C03626=1136.287,55.628,-52.348,-179.813,6.522,149.136
C03627=1136.292,55.380,-52.331,-179.816,6.520,149.137
C03628=1136.297,55.129,-52.315,-179.818,6.519,149.137
C03629=1136.302,54.880,-52.300,-179.821,6.518,149.138
C03630=1136.307,54.631,-52.285,-179.824,6.516,149.138
C03631=1136.312,54.381,-52.269,-179.826,6.515,149.139
C03632=1136.317,54.132,-52.253,-179.829,6.514,149.139
C03633=1136.322,53.883,-52.237,-179.831,6.513,149.140
C03634=1136.327,53.613,-52.220,-179.834,6.512,149.140
C03635=1136.333,53.345,-52.203,-179.837,6.510,149.141
C03636=1136.338,53.076,-52.187,-179.840,6.509,149.142
C03637=1136.343,52.808,-52.170,-179.843,6.507,149.142
C03638=1136.349,52.558,-52.154,-179.846,6.507,149.143
C03639=1136.353,52.309,-52.138,-179.848,6.505,149.143
C03640=1136.358,52.059,-52.122,-179.850,6.504,149.144
C03641=1136.363,51.810,-52.107,-179.854,6.503,149.144
C03642=1136.369,51.561,-52.091,-179.856,6.502,149.145
C03643=1136.373,51.311,-52.075,-179.859,6.500,149.145
C03644=1136.379,51.061,-52.060,-179.862,6.499,149.146
C03645=1136.383,50.812,-52.045,-179.864,6.498,149.146
C03646=1136.388,50.562,-52.029,-179.867,6.497,149.147
C03647=1136.394,50.313,-52.013,-179.869,6.496,149.147
C03648=1136.399,50.063,-51.998,-179.872,6.495,149.148
C03649=1136.404,49.814,-51.983,-179.874,6.494,149.148
C03650=1136.408,49.564,-51.967,-179.878,6.492,149.149
C03651=1136.414,49.315,-51.951,-179.880,6.491,149.149
C03652=1136.418,49.066,-51.936,-179.882,6.490,149.150
C03653=1136.424,48.816,-51.921,-179.885,6.488,149.150
C03654=1136.429,48.567,-51.905,-179.888,6.488,149.151
C03655=1136.433,48.317,-51.890,-179.891,6.486,149.151
C03656=1136.439,48.068,-51.874,-179.893,6.485,149.152
C03657=1136.444,47.818,-51.858,-179.896,6.484,149.152
C03658=1136.449,47.569,-51.843,-179.898,6.483,149.153
C03659=1136.453,47.319,-51.828,-179.901,6.482,149.153
C03660=1136.459,47.070,-51.812,-179.904,6.480,149.154
C03661=1136.463,46.821,-51.797,-179.906,6.480,149.154
C03662=1136.469,46.571,-51.781,-179.909,6.478,149.155
C03663=1136.473,46.322,-51.766,-179.912,6.478,149.156
C03664=1136.479,46.073,-51.751,-179.915,6.476,149.156
C03665=1136.484,45.822,-51.736,-179.917,6.475,149.156
C03666=1136.489,45.573,-51.721,-179.919,6.473,149.157
C03667=1136.494,45.324,-51.705,-179.922,6.473,149.158
C03668=1136.499,45.074,-51.690,-179.925,6.471,149.158
C03669=1136.504,44.825,-51.674,-179.927,6.470,149.158
C03670=1136.509,44.576,-51.659,-179.930,6.469,149.159
C03671=1136.514,44.325,-51.644,-179.932,6.468,149.160
C03672=1136.519,44.076,-51.629,-179.935,6.467,149.160
C03673=1136.524,43.827,-51.614,-179.938,6.466,149.161
C03674=1136.529,43.577,-51.598,-179.941,6.465,149.161
C03675=1136.534,43.328,-51.583,-179.943,6.464,149.162
C03676=1136.540,43.078,-51.568,-179.946,6.463,149.162
C03677=1136.544,42.829,-51.553,-179.949,6.461,149.163
C03678=1136.549,42.579,-51.537,-179.951,6.460,149.163
C03679=1136.554,42.330,-51.522,-179.954,6.459,149.164
C03680=1136.559,42.080,-51.507,-179.956,6.458,149.164
C03681=1136.564,41.831,-51.492,-179.959,6.456,149.165
C03682=1136.569,41.581,-51.477,-179.962,6.456,149.165
C03683=1136.574,41.332,-51.462,-179.964,6.454,149.166
C03684=1136.580,41.082,-51.447,-179.967,6.454,149.166
C03685=1136.584,40.833,-51.432,-179.970,6.452,149.167
C03686=1136.590,40.583,-51.417,-179.972,6.451,149.167
C03687=1136.595,40.334,-51.402,-179.975,6.450,149.168
C03688=1136.600,40.085,-51.386,-179.977,6.449,149.169
C03689=1136.605,39.835,-51.372,-179.980,6.448,149.169
C03690=1136.610,39.585,-51.356,-179.982,6.447,149.169
C03691=1136.614,39.336,-51.341,-179.985,6.445,149.170
C03692=1136.619,39.086,-51.327,-179.988,6.445,149.171
C03693=1136.625,38.837,-51.311,-179.990,6.444,149.171
C03694=1136.630,38.587,-51.297,-179.993,6.442,149.171
C03695=1136.635,38.338,-51.281,-179.995,6.442,149.172
C03696=1136.640,38.088,-51.266,-179.998,6.440,149.173
C03697=1136.645,37.839,-51.252,180.000,6.439,149.173
C03698=1136.650,37.589,-51.237,179.996,6.438,149.174
C03699=1136.655,37.340,-51.222,179.994,6.437,149.174
C03700=1136.660,37.090,-51.207,179.992,6.436,149.175
C03701=1136.665,36.841,-51.192,179.989,6.435,149.175
C03702=1136.670,36.591,-51.177,179.986,6.434,149.176
C03703=1136.676,36.341,-51.163,179.984,6.433,149.176
C03704=1136.680,36.092,-51.148,179.981,6.432,149.177
C03705=1136.685,35.843,-51.133,179.979,6.431,149.177
C03706=1136.691,35.593,-51.118,179.976,6.429,149.178
C03707=1136.696,35.343,-51.103,179.973,6.429,149.178
C03708=1136.700,35.094,-51.088,179.970,6.427,149.179
C03709=1136.706,34.844,-51.074,179.968,6.426,149.179
C03710=1136.711,34.595,-51.059,179.966,6.426,149.180
C03711=1136.716,34.346,-51.044,179.963,6.424,149.180
C03712=1136.721,34.096,-51.029,179.961,6.423,149.181
C03713=1136.726,33.846,-51.014,179.957,6.422,149.182
C03714=1136.731,33.597,-51.000,179.955,6.421,149.182
C03715=1136.736,33.348,-50.985,179.952,6.420,149.183
C03716=1136.742,33.098,-50.971,179.950,6.419,149.183
C03717=1136.747,32.849,-50.956,179.947,6.418,149.184
C03718=1136.751,32.600,-50.941,179.945,6.417,149.184
C03719=1136.756,32.350,-50.927,179.942,6.416,149.185
C03720=1136.762,32.100,-50.912,179.939,6.415,149.185
C03721=1136.767,31.851,-50.897,179.937,6.414,149.186
C03722=1136.772,31.601,-50.883,179.934,6.413,149.186
C03723=1136.777,31.351,-50.869,179.932,6.412,149.187
C03724=1136.782,31.102,-50.853,179.929,6.411,149.187
C03725=1136.787,30.852,-50.839,179.926,6.410,149.188
C03726=1136.792,30.602,-50.825,179.924,6.409,149.188
C03727=1136.797,30.353,-50.810,179.921,6.408,149.189
C03728=1136.802,30.104,-50.796,179.919,6.407,149.190
C03729=1136.808,29.854,-50.781,179.916,6.405,149.190
C03730=1136.813,29.605,-50.767,179.914,6.405,149.191
C03731=1136.817,29.356,-50.752,179.911,6.403,149.191
C03732=1136.822,29.106,-50.737,179.909,6.402,149.192
C03733=1136.827,28.856,-50.723,179.906,6.402,149.192
C03734=1136.832,28.606,-50.709,179.903,6.400,149.193
C03735=1136.837,28.357,-50.694,179.901,6.399,149.193
C03736=1136.843,28.108,-50.679,179.898,6.398,149.194
C03737=1136.848,27.858,-50.665,179.896,6.397,149.194
C03738=1136.853,27.590,-50.649,179.893,6.396,149.195
C03739=1136.859,27.320,-50.634,179.890,6.395,149.195
C03740=1136.864,27.051,-50.619,179.887,6.394,149.196
C03741=1136.870,26.782,-50.602,179.885,6.393,149.197
C03742=1136.875,26.532,-50.588,179.882,6.392,149.197
C03743=1136.880,26.283,-50.574,179.879,6.391,149.198
C03744=1136.885,26.034,-50.560,179.877,6.390,149.198
C03745=1136.890,25.784,-50.545,179.874,6.389,149.199
C03746=1136.895,25.534,-50.531,179.872,6.388,149.199
C03747=1136.900,25.285,-50.517,179.869,6.387,149.200
C03748=1136.905,25.035,-50.503,179.866,6.386,149.200
C03749=1136.911,24.786,-50.489,179.864,6.385,149.201
C03750=1136.916,24.536,-50.474,179.861,6.384,149.201
C03751=1136.921,24.286,-50.460,179.859,6.383,149.202
C03752=1136.925,24.037,-50.445,179.856,6.382,149.202
C03753=1136.930,23.788,-50.431,179.854,6.381,149.203
C03754=1136.936,23.539,-50.417,179.851,6.381,149.204
C03755=1136.941,23.289,-50.403,179.848,6.379,149.204
C03756=1136.946,23.039,-50.388,179.846,6.378,149.205
C03757=1136.951,22.790,-50.374,179.843,6.377,149.205
C03758=1136.956,22.541,-50.360,179.841,6.376,149.206
C03759=1136.961,22.291,-50.346,179.839,6.375,149.206
C03760=1136.966,22.041,-50.332,179.835,6.374,149.207
C03761=1136.971,21.791,-50.317,179.833,6.373,149.207
C03762=1136.977,21.542,-50.304,179.831,6.372,149.208
C03763=1136.982,21.292,-50.290,179.828,6.371,149.208
C03764=1136.987,21.042,-50.276,179.826,6.370,149.209
C03765=1136.992,20.793,-50.261,179.823,6.369,149.209
C03766=1136.997,20.544,-50.247,179.820,6.368,149.210
C03767=1137.002,20.294,-50.233,179.818,6.367,149.210
C03768=1137.007,20.044,-50.219,179.815,6.366,149.211
C03769=1137.013,19.795,-50.205,179.813,6.365,149.212
C03770=1137.018,19.546,-50.191,179.810,6.365,149.212
C03771=1137.023,19.296,-50.176,179.807,6.363,149.213
C03772=1137.027,19.046,-50.163,179.805,6.362,149.213
C03773=1137.033,18.797,-50.150,179.803,6.362,149.214
C03774=1137.038,18.547,-50.135,179.800,6.360,149.214
C03775=1137.043,18.297,-50.121,179.797,6.360,149.215
C03776=1137.048,18.048,-50.107,179.795,6.359,149.215
C03777=1137.053,17.799,-50.093,179.792,6.358,149.216
C03778=1137.058,17.549,-50.079,179.790,6.357,149.216
C03779=1137.064,17.299,-50.065,179.788,6.356,149.217
C03780=1137.068,17.050,-50.052,179.784,6.355,149.218
C03781=1137.073,16.800,-50.037,179.782,6.354,149.218
C03782=1137.079,16.551,-50.024,179.780,6.353,149.219
C03783=1137.084,16.301,-50.009,179.777,6.352,149.219
C03784=1137.089,16.051,-49.996,179.775,6.351,149.220
C03785=1137.094,15.802,-49.982,179.772,6.351,149.220
C03786=1137.099,15.553,-49.968,179.769,6.349,149.221
C03787=1137.104,15.302,-49.955,179.767,6.348,149.221
C03788=1137.109,15.053,-49.941,179.764,6.348,149.222
C03789=1137.114,14.804,-49.926,179.762,6.346,149.222
C03790=1137.119,14.554,-49.912,179.759,6.345,149.223
C03791=1137.125,14.305,-49.899,179.757,6.345,149.223
C03792=1137.129,14.055,-49.885,179.754,6.343,149.224
C03793=1137.135,13.806,-49.871,179.752,6.342,149.224
C03794=1137.140,13.556,-49.858,179.749,6.342,149.225
C03795=1137.145,13.306,-49.844,179.747,6.341,149.226
C03796=1137.150,13.057,-49.830,179.744,6.340,149.226
C03797=1137.155,12.807,-49.817,179.742,6.339,149.227
C03798=1137.161,12.558,-49.803,179.739,6.338,149.227
C03799=1137.165,12.308,-49.789,179.736,6.337,149.228
C03800=1137.170,12.058,-49.775,179.734,6.336,149.228
C03801=1137.176,11.809,-49.761,179.732,6.336,149.229
C03802=1137.180,11.559,-49.749,179.729,6.334,149.229
C03803=1137.186,11.310,-49.735,179.726,6.333,149.230
C03804=1137.191,11.060,-49.720,179.724,6.333,149.230
C03805=1137.197,10.811,-49.707,179.722,6.332,149.231
C03806=1137.201,10.561,-49.693,179.719,6.331,149.232
C03807=1137.206,10.311,-49.680,179.716,6.330,149.232
C03808=1137.212,10.062,-49.666,179.714,6.329,149.233
C03809=1137.216,9.812,-49.653,179.711,6.328,149.233
C03810=1137.222,9.563,-49.639,179.709,6.327,149.234
C03811=1137.227,9.313,-49.626,179.706,6.327,149.234
C03812=1137.232,9.064,-49.612,179.704,6.326,149.235
C03813=1137.237,8.814,-49.599,179.701,6.325,149.235
C03814=1137.243,8.565,-49.585,179.699,6.324,149.236
C03815=1137.247,8.315,-49.572,179.697,6.323,149.236
C03816=1137.253,8.066,-49.558,179.693,6.322,149.237
C03817=1137.257,7.816,-49.545,179.691,6.321,149.237
C03818=1137.263,7.567,-49.531,179.688,6.320,149.238
C03819=1137.268,7.316,-49.517,179.686,6.320,149.239
C03820=1137.273,7.068,-49.504,179.684,6.318,149.239
C03821=1137.278,6.817,-49.491,179.681,6.318,149.240
C03822=1137.283,6.568,-49.478,179.679,6.317,149.240
C03823=1137.288,6.318,-49.464,179.677,6.316,149.241
C03824=1137.294,6.069,-49.450,179.673,6.315,149.241
C03825=1137.298,5.819,-49.437,179.671,6.314,149.242
C03826=1137.304,5.570,-49.424,179.669,6.313,149.242
C03827=1137.309,5.319,-49.411,179.666,6.313,149.243
C03828=1137.314,5.070,-49.397,179.664,6.311,149.243
C03829=1137.319,4.820,-49.384,179.661,6.311,149.244
C03830=1137.325,4.571,-49.371,179.659,6.310,149.245
C03831=1137.329,4.321,-49.357,179.657,6.309,149.245
C03832=1137.335,4.072,-49.344,179.653,6.308,149.246
C03833=1137.339,3.822,-49.331,179.651,6.307,149.246
C03834=1137.345,3.573,-49.317,179.649,6.306,149.247
C03835=1137.350,3.323,-49.304,179.646,6.306,149.247
C03836=1137.355,3.073,-49.291,179.643,6.304,149.248
C03837=1137.360,2.824,-49.277,179.641,6.303,149.248
C03838=1137.365,2.574,-49.264,179.639,6.303,149.249
C03839=1137.371,2.325,-49.251,179.636,6.302,149.249
C03840=1137.376,2.074,-49.238,179.633,6.301,149.250
C03841=1137.381,1.826,-49.224,179.631,6.300,149.251
C03842=1137.386,1.556,-49.210,179.629,6.299,149.251
C03843=1137.393,1.286,-49.196,179.626,6.298,149.252
C03844=1137.397,1.017,-49.182,179.623,6.298,149.252
C03845=1137.403,0.747,-49.167,179.621,6.297,149.253
C03846=1137.408,0.498,-49.155,179.618,6.295,149.253
C03847=1137.413,0.248,-49.141,179.615,6.295,149.254
C03848=1137.418,-0.001,-49.128,179.613,6.294,149.255
C03849=1137.424,-0.251,-49.115,179.610,6.294,149.255
C03850=1137.429,-0.501,-49.102,179.608,6.293,149.256
C03851=1137.434,-0.750,-49.089,179.606,6.291,149.256
C03852=1137.440,-1.000,-49.076,179.603,6.291,149.257
C03853=1137.444,-1.249,-49.062,179.601,6.290,149.257
C03854=1137.450,-1.499,-49.049,179.599,6.289,149.258
C03855=1137.454,-1.749,-49.036,179.595,6.288,149.258
C03856=1137.459,-1.998,-49.024,179.593,6.287,149.259
C03857=1137.465,-2.248,-49.010,179.591,6.286,149.259
C03858=1137.470,-2.498,-48.997,179.588,6.286,149.260
C03859=1137.475,-2.747,-48.985,179.586,6.285,149.261
C03860=1137.481,-2.997,-48.972,179.583,6.284,149.261
C03861=1137.485,-3.247,-48.959,179.581,6.283,149.262
C03862=1137.491,-3.496,-48.945,179.578,6.282,149.262
C03863=1137.496,-3.745,-48.932,179.576,6.282,149.263
C03864=1137.501,-3.995,-48.919,179.574,6.281,149.263
C03865=1137.506,-4.244,-48.907,179.571,6.280,149.264
C03866=1137.512,-4.494,-48.893,179.568,6.279,149.265
C03867=1137.517,-4.743,-48.881,179.566,6.278,149.265
C03868=1137.521,-4.993,-48.868,179.564,6.278,149.265
C03869=1137.527,-5.243,-48.855,179.561,6.277,149.266
C03870=1137.532,-5.492,-48.842,179.559,6.276,149.267
C03871=1137.537,-5.742,-48.829,179.556,6.275,149.267
C03872=1137.543,-5.992,-48.816,179.554,6.274,149.268
C03873=1137.548,-6.241,-48.803,179.551,6.273,149.268
C03874=1137.553,-6.491,-48.791,179.549,6.273,149.269
C03875=1137.557,-6.741,-48.778,179.547,6.272,149.269
C03876=1137.563,-6.990,-48.764,179.544,6.271,149.270
C03877=1137.569,-7.240,-48.753,179.541,6.270,149.271
C03878=1137.573,-7.490,-48.740,179.539,6.269,149.271
C03879=1137.578,-7.739,-48.727,179.537,6.269,149.271
C03880=1137.584,-7.989,-48.714,179.534,6.268,149.272
C03881=1137.589,-8.238,-48.701,179.532,6.267,149.273
C03882=1137.594,-8.488,-48.688,179.529,6.267,149.273
C03883=1137.599,-8.738,-48.676,179.526,6.265,149.274
C03884=1137.604,-8.987,-48.663,179.524,6.265,149.274
C03885=1137.610,-9.237,-48.650,179.522,6.264,149.275
C03886=1137.614,-9.487,-48.637,179.519,6.263,149.275
C03887=1137.620,-9.737,-48.625,179.517,6.263,149.276
C03888=1137.625,-9.986,-48.612,179.515,6.262,149.277
C03889=1137.630,-10.235,-48.600,179.512,6.261,149.277
C03890=1137.635,-10.485,-48.587,179.510,6.260,149.278
C03891=1137.640,-10.735,-48.574,179.507,6.259,149.278
C03892=1137.646,-10.984,-48.561,179.505,6.259,149.279
C03893=1137.651,-11.234,-48.549,179.502,6.258,149.279
C03894=1137.656,-11.483,-48.537,179.500,6.257,149.280
C03895=1137.661,-11.733,-48.524,179.498,6.257,149.280
C03896=1137.666,-11.983,-48.511,179.495,6.255,149.281
C03897=1137.671,-12.232,-48.498,179.492,6.255,149.281
C03898=1137.677,-12.482,-48.486,179.490,6.254,149.282
C03899=1137.682,-12.732,-48.473,179.488,6.253,149.283
C03900=1137.687,-12.981,-48.461,179.485,6.253,149.283
C03901=1137.692,-13.231,-48.448,179.483,6.252,149.284
C03902=1137.697,-13.481,-48.436,179.480,6.251,149.284
C03903=1137.702,-13.730,-48.423,179.478,6.251,149.285
C03904=1137.708,-13.980,-48.411,179.476,6.249,149.285
C03905=1137.713,-14.230,-48.399,179.473,6.249,149.286
C03906=1137.718,-14.479,-48.386,179.471,6.248,149.286
C03907=1137.723,-14.728,-48.374,179.468,6.247,149.287
C03908=1137.728,-14.979,-48.361,179.466,6.247,149.288
C03909=1137.733,-15.228,-48.349,179.464,6.246,149.288
C03910=1137.739,-15.478,-48.335,179.461,6.245,149.289
C03911=1137.744,-15.728,-48.324,179.459,6.245,149.289
C03912=1137.750,-15.977,-48.311,179.456,6.243,149.290
C03913=1137.755,-16.226,-48.298,179.453,6.243,149.290
C03914=1137.760,-16.476,-48.287,179.451,6.242,149.291
C03915=1137.765,-16.726,-48.274,179.449,6.241,149.291
C03916=1137.770,-16.976,-48.261,179.446,6.241,149.292
C03917=1137.775,-17.226,-48.249,179.444,6.240,149.292
C03918=1137.780,-17.475,-48.236,179.442,6.239,149.293
C03919=1137.786,-17.725,-48.225,179.439,6.239,149.294
C03920=1137.791,-17.974,-48.212,179.437,6.238,149.294
C03921=1137.796,-18.223,-48.199,179.434,6.237,149.295
C03922=1137.801,-18.473,-48.188,179.432,6.236,149.295
C03923=1137.807,-18.723,-48.175,179.430,6.235,149.296
C03924=1137.812,-18.973,-48.163,179.427,6.235,149.296
C03925=1137.817,-19.222,-48.150,179.425,6.234,149.297
C03926=1137.823,-19.472,-48.139,179.422,6.233,149.297
C03927=1137.827,-19.722,-48.126,179.420,6.233,149.298
C03928=1137.832,-19.972,-48.114,179.418,6.232,149.299
C03929=1137.837,-20.221,-48.102,179.415,6.231,149.299
C03930=1137.842,-20.471,-48.090,179.413,6.231,149.300
C03931=1137.847,-20.720,-48.077,179.411,6.230,149.300
C03932=1137.853,-20.970,-48.065,179.408,6.229,149.301
C03933=1137.858,-21.219,-48.053,179.405,6.228,149.301
C03934=1137.863,-21.469,-48.041,179.403,6.227,149.302
C03935=1137.869,-21.719,-48.028,179.400,6.227,149.302
C03936=1137.874,-21.969,-48.016,179.398,6.226,149.303
C03937=1137.879,-22.218,-48.004,179.396,6.225,149.303
C03938=1137.885,-22.468,-47.992,179.393,6.225,149.304
C03939=1137.890,-22.718,-47.980,179.391,6.224,149.305
C03940=1137.894,-22.967,-47.968,179.389,6.223,149.305
C03941=1137.900,-23.217,-47.956,179.386,6.223,149.306
C03942=1137.905,-23.466,-47.943,179.384,6.222,149.306
C03943=1137.910,-23.716,-47.932,179.382,6.221,149.307
C03944=1137.916,-23.966,-47.920,179.379,6.221,149.307
C03945=1137.921,-24.215,-47.907,179.377,6.220,149.308
C03946=1137.926,-24.486,-47.894,179.374,6.219,149.309
C03947=1137.932,-24.755,-47.882,179.372,6.218,149.309
C03948=1137.937,-25.026,-47.869,179.369,6.217,149.310
C03949=1137.943,-25.296,-47.855,179.367,6.217,149.310
C03950=1137.948,-25.545,-47.843,179.364,6.216,149.311
C03951=1137.954,-25.794,-47.831,179.362,6.215,149.311
C03952=1137.959,-26.044,-47.820,179.360,6.215,149.312
C03953=1137.965,-26.294,-47.808,179.356,6.213,149.313
C03954=1137.969,-26.543,-47.796,179.354,6.213,149.313
C03955=1137.975,-26.793,-47.784,179.352,6.212,149.314
C03956=1137.980,-27.043,-47.772,179.349,6.212,149.314
C03957=1137.985,-27.293,-47.759,179.347,6.211,149.315
C03958=1137.991,-27.542,-47.747,179.345,6.210,149.315
C03959=1137.995,-27.792,-47.736,179.342,6.210,149.316
C03960=1138.001,-28.042,-47.724,179.340,6.209,149.316
C03961=1138.006,-28.291,-47.712,179.338,6.208,149.317
C03962=1138.011,-28.541,-47.700,179.335,6.208,149.318
C03963=1138.016,-28.791,-47.688,179.333,6.207,149.318
C03964=1138.021,-29.041,-47.677,179.331,6.206,149.318
C03965=1138.026,-29.290,-47.664,179.328,6.206,149.319
C03966=1138.031,-29.540,-47.653,179.326,6.205,149.320
C03967=1138.037,-29.790,-47.641,179.324,6.204,149.320
C03968=1138.043,-30.039,-47.629,179.321,6.204,149.321
C03969=1138.048,-30.289,-47.617,179.319,6.203,149.321
C03970=1138.053,-30.539,-47.606,179.317,6.202,149.322
C03971=1138.058,-30.788,-47.594,179.314,6.202,149.322
C03972=1138.063,-31.038,-47.582,179.312,6.201,149.323
C03973=1138.068,-31.287,-47.570,179.310,6.200,149.323
C03974=1138.073,-31.537,-47.558,179.307,6.200,149.324
C03975=1138.079,-31.787,-47.547,179.305,6.199,149.325
C03976=1138.083,-32.037,-47.535,179.303,6.198,149.325
C03977=1138.090,-32.286,-47.524,179.300,6.198,149.326
C03978=1138.095,-32.535,-47.511,179.298,6.197,149.326
C03979=1138.099,-32.785,-47.500,179.296,6.196,149.327
C03980=1138.105,-33.035,-47.488,179.293,6.196,149.327
C03981=1138.110,-33.285,-47.476,179.291,6.195,149.328
C03982=1138.115,-33.535,-47.465,179.288,6.195,149.329
C03983=1138.120,-33.785,-47.453,179.286,6.194,149.329
C03984=1138.126,-34.034,-47.441,179.284,6.193,149.330
C03985=1138.131,-34.283,-47.430,179.281,6.193,149.330
C03986=1138.136,-34.533,-47.418,179.279,6.192,149.331
C03987=1138.141,-34.783,-47.407,179.277,6.191,149.331
C03988=1138.147,-35.033,-47.395,179.274,6.191,149.332
C03989=1138.152,-35.283,-47.383,179.272,6.190,149.332
C03990=1138.157,-35.532,-47.372,179.270,6.189,149.333
C03991=1138.163,-35.782,-47.360,179.267,6.189,149.334
C03992=1138.167,-36.031,-47.349,179.265,6.188,149.334
C03993=1138.173,-36.281,-47.337,179.263,6.187,149.334
C03994=1138.178,-36.531,-47.326,179.260,6.187,149.335
C03995=1138.184,-36.780,-47.314,179.258,6.186,149.336
C03996=1138.189,-37.030,-47.303,179.256,6.185,149.336
C03997=1138.194,-37.280,-47.291,179.253,6.185,149.337
C03998=1138.199,-37.530,-47.279,179.251,6.184,149.337
C03999=1138.204,-37.779,-47.268,179.249,6.183,149.338
C04000=1138.210,-38.028,-47.257,179.247,6.182,149.338
C04001=1138.215,-38.278,-47.245,179.244,6.182,149.339
C04002=1138.220,-38.528,-47.233,179.242,6.181,149.339
C04003=1138.225,-38.778,-47.222,179.240,6.180,149.340
C04004=1138.231,-39.027,-47.211,179.237,6.180,149.341
C04005=1138.236,-39.277,-47.200,179.235,6.179,149.341
C04006=1138.241,-39.527,-47.188,179.232,6.178,149.342
C04007=1138.246,-39.777,-47.177,179.230,6.178,149.342
C04008=1138.252,-40.026,-47.165,179.228,6.177,149.343
C04009=1138.257,-40.276,-47.154,179.225,6.176,149.343
C04010=1138.262,-40.525,-47.142,179.223,6.176,149.344
C04011=1138.267,-40.775,-47.131,179.221,6.175,149.344
C04012=1138.273,-41.025,-47.120,179.218,6.175,149.345
C04013=1138.278,-41.275,-47.109,179.216,6.174,149.346
C04014=1138.283,-41.525,-47.097,179.214,6.173,149.346
C04015=1138.288,-41.774,-47.086,179.211,6.173,149.347
C04016=1138.294,-42.023,-47.074,179.209,6.173,149.347
C04017=1138.299,-42.273,-47.063,179.207,6.172,149.348
C04018=1138.304,-42.523,-47.052,179.205,6.171,149.348
C04019=1138.310,-42.772,-47.041,179.202,6.171,149.349
C04020=1138.314,-43.022,-47.029,179.200,6.170,149.349
C04021=1138.320,-43.272,-47.017,179.198,6.169,149.350
C04022=1138.325,-43.522,-47.007,179.195,6.169,149.351
C04023=1138.331,-43.772,-46.995,179.193,6.168,149.351
C04024=1138.335,-44.021,-46.984,179.191,6.168,149.351
C04025=1138.340,-44.271,-46.973,179.188,6.167,149.352
C04026=1138.346,-44.521,-46.962,179.186,6.166,149.353
C04027=1138.351,-44.770,-46.951,179.184,6.166,149.353
C04028=1138.356,-45.020,-46.939,179.182,6.165,149.354
C04029=1138.362,-45.269,-46.928,179.179,6.164,149.354
C04030=1138.367,-45.519,-46.917,179.177,6.164,149.355
C04031=1138.372,-45.769,-46.905,179.175,6.163,149.355
C04032=1138.378,-46.018,-46.895,179.172,6.162,149.356
C04033=1138.383,-46.268,-46.884,179.170,6.162,149.356
C04034=1138.388,-46.518,-46.872,179.168,6.162,149.357
C04035=1138.393,-46.767,-46.861,179.165,6.161,149.358
C04036=1138.398,-47.018,-46.851,179.163,6.161,149.358
C04037=1138.404,-47.268,-46.839,179.161,6.160,149.359
C04038=1138.409,-47.516,-46.828,179.158,6.159,149.359
C04039=1138.414,-47.767,-46.817,179.156,6.159,149.360
C04040=1138.419,-48.017,-46.805,179.154,6.158,149.360
C04041=1138.425,-48.266,-46.795,179.151,6.157,149.361
C04042=1138.430,-48.516,-46.784,179.149,6.157,149.361
C04043=1138.436,-48.765,-46.772,179.147,6.156,149.362
C04044=1138.441,-49.015,-46.762,179.145,6.155,149.362
C04045=1138.445,-49.265,-46.750,179.143,6.155,149.363
C04046=1138.451,-49.514,-46.740,179.141,6.155,149.364
C04047=1138.456,-49.764,-46.728,179.138,6.154,149.364
C04048=1138.462,-50.013,-46.717,179.136,6.154,149.365
C04049=1138.467,-50.264,-46.707,179.134,6.153,149.365
C04050=1138.472,-50.535,-46.695,179.131,6.152,149.366
C04051=1138.479,-50.805,-46.683,179.129,6.152,149.366
C04052=1138.484,-51.076,-46.670,179.126,6.151,149.367
C04053=1138.489,-51.347,-46.659,179.124,6.150,149.368
C04054=1138.495,-51.596,-46.648,179.122,6.150,149.368
C04055=1138.500,-51.846,-46.637,179.119,6.149,149.369
C04056=1138.506,-52.095,-46.626,179.117,6.149,149.369
C04057=1138.510,-52.345,-46.615,179.115,6.148,149.370
C04058=1138.515,-52.595,-46.605,179.112,6.147,149.370
C04059=1138.522,-52.845,-46.594,179.110,6.147,149.371
C04060=1138.526,-53.095,-46.582,179.107,6.146,149.371
C04061=1138.532,-53.344,-46.572,179.106,6.146,149.372
C04062=1138.537,-53.594,-46.561,179.103,6.145,149.373
C04063=1138.542,-53.844,-46.551,179.101,6.145,149.373
C04064=1138.548,-54.093,-46.539,179.099,6.144,149.374
C04065=1138.553,-54.343,-46.529,179.096,6.144,149.374
C04066=1138.558,-54.593,-46.517,179.094,6.143,149.375
C04067=1138.564,-54.842,-46.507,179.092,6.142,149.375
C04068=1138.569,-55.092,-46.497,179.090,6.141,149.376
C04069=1138.573,-55.342,-46.485,179.088,6.142,149.376
C04070=1138.579,-55.592,-46.475,179.085,6.141,149.377
C04071=1138.584,-55.842,-46.463,179.083,6.140,149.377
C04072=1138.590,-56.091,-46.453,179.080,6.140,149.378
C04073=1138.595,-56.341,-46.442,179.078,6.139,149.379
C04074=1138.600,-56.590,-46.432,179.076,6.138,149.379
C04075=1138.605,-56.840,-46.421,179.074,6.137,149.379
C04076=1138.611,-57.090,-46.411,179.071,6.137,149.380
C04077=1138.616,-57.340,-46.399,179.070,6.137,149.381
C04078=1138.621,-57.589,-46.389,179.067,6.136,149.381
C04079=1138.626,-57.839,-46.379,179.065,6.136,149.382
C04080=1138.631,-58.088,-46.368,179.063,6.135,149.382
C04081=1138.637,-58.339,-46.357,179.060,6.134,149.383
C04082=1138.643,-58.588,-46.346,179.058,6.134,149.383
C04083=1138.647,-58.838,-46.335,179.056,6.133,149.384
C04084=1138.653,-59.088,-46.325,179.054,6.133,149.384
C04085=1138.658,-59.338,-46.314,179.052,6.132,149.385
C04086=1138.663,-59.587,-46.303,179.050,6.132,149.385
C04087=1138.668,-59.837,-46.293,179.047,6.131,149.386
C04088=1138.674,-60.087,-46.283,179.045,6.130,149.387
C04089=1138.680,-60.336,-46.272,179.043,6.130,149.387
C04090=1138.684,-60.586,-46.261,179.040,6.129,149.388
C04091=1138.690,-60.835,-46.251,179.038,6.129,149.388
C04092=1138.695,-61.086,-46.240,179.036,6.129,149.389
C04093=1138.700,-61.335,-46.230,179.034,6.128,149.389
C04094=1138.705,-61.585,-46.219,179.031,6.127,149.390
C04095=1138.711,-61.834,-46.209,179.029,6.127,149.390
C04096=1138.716,-62.085,-46.198,179.027,6.126,149.391
C04097=1138.721,-62.334,-46.188,179.025,6.126,149.392
C04098=1138.727,-62.584,-46.178,179.023,6.126,149.392
C04099=1138.732,-62.833,-46.166,179.020,6.125,149.393
C04100=1138.737,-63.083,-46.156,179.018,6.124,149.393
C04101=1138.742,-63.333,-46.146,179.016,6.124,149.394
C04102=1138.748,-63.583,-46.135,179.013,6.123,149.394
C04103=1138.753,-63.833,-46.125,179.012,6.123,149.395
C04104=1138.758,-64.082,-46.115,179.010,6.122,149.395
C04105=1138.764,-64.332,-46.104,179.007,6.122,149.396
C04106=1138.769,-64.582,-46.093,179.005,6.121,149.396
C04107=1138.774,-64.831,-46.083,179.003,6.120,149.397
C04108=1138.779,-65.081,-46.072,179.001,6.120,149.397
C04109=1138.785,-65.331,-46.062,178.998,6.120,149.398
C04110=1138.790,-65.580,-46.052,178.996,6.119,149.399
C04111=1138.795,-65.831,-46.041,178.994,6.118,149.399
C04112=1138.801,-66.080,-46.031,178.992,6.117,149.399
C04113=1138.806,-66.329,-46.021,178.989,6.117,149.400
C04114=1138.811,-66.580,-46.011,178.987,6.117,149.401
C04115=1138.817,-66.829,-46.001,178.985,6.116,149.401
C04116=1138.822,-67.079,-45.990,178.983,6.116,149.402
C04117=1138.827,-67.328,-45.979,178.980,6.115,149.402
C04118=1138.832,-67.578,-45.969,178.978,6.114,149.403
C04119=1138.837,-67.828,-45.958,178.977,6.114,149.403
C04120=1138.843,-68.078,-45.948,178.974,6.114,149.404
C04121=1138.849,-68.327,-45.938,178.972,6.113,149.405
C04122=1138.853,-68.577,-45.928,178.970,6.113,149.405
C04123=1138.858,-68.827,-45.918,178.967,6.112,149.405
C04124=1138.864,-69.076,-45.908,178.966,6.112,149.406
C04125=1138.869,-69.327,-45.897,178.963,6.111,149.407
C04126=1138.875,-69.576,-45.887,178.961,6.111,149.407
C04127=1138.880,-69.826,-45.877,178.959,6.110,149.408
C04128=1138.886,-70.075,-45.866,178.956,6.109,149.408
C04129=1138.890,-70.325,-45.856,178.954,6.110,149.409
C04130=1138.896,-70.575,-45.847,178.952,6.109,149.409
C04131=1138.902,-70.825,-45.837,178.950,6.108,149.410
C04132=1138.907,-71.075,-45.826,178.948,6.107,149.410
C04133=1138.912,-71.325,-45.816,178.945,6.107,149.411
C04134=1138.918,-71.574,-45.806,178.944,6.107,149.411
C04135=1138.922,-71.824,-45.796,178.941,6.106,149.412
C04136=1138.928,-72.074,-45.786,178.939,6.105,149.412
C04137=1138.933,-72.323,-45.775,178.937,6.105,149.413
C04138=1138.939,-72.573,-45.765,178.935,6.105,149.414
C04139=1138.944,-72.823,-45.755,178.933,6.104,149.414
C04140=1138.949,-73.072,-45.745,178.931,6.104,149.415
C04141=1138.954,-73.322,-45.735,178.928,6.103,149.415
C04142=1138.960,-73.572,-45.725,178.926,6.102,149.416
C04143=1138.965,-73.822,-45.715,178.924,6.102,149.416
C04144=1138.971,-74.072,-45.704,178.922,6.102,149.417
C04145=1138.976,-74.321,-45.695,178.919,6.101,149.417
C04146=1138.981,-74.570,-45.685,178.917,6.101,149.418
C04147=1138.986,-74.821,-45.674,178.915,6.101,149.418
C04148=1138.992,-75.071,-45.665,178.913,6.100,149.419
C04149=1138.997,-75.320,-45.655,178.911,6.099,149.419
C04150=1139.003,-75.570,-45.645,178.908,6.099,149.420
C04151=1139.008,-75.820,-45.634,178.907,6.099,149.421
C04152=1139.013,-76.069,-45.624,178.905,6.098,149.421
C04153=1139.018,-76.319,-45.615,178.902,6.097,149.422
C04154=1139.024,-76.591,-45.603,178.900,6.097,149.422
C04155=1139.030,-76.862,-45.593,178.898,6.096,149.423
C04156=1139.036,-77.134,-45.582,178.895,6.096,149.423
C04157=1139.042,-77.405,-45.571,178.893,6.095,149.424
C04158=1139.047,-77.655,-45.561,178.891,6.095,149.424
C04159=1139.052,-77.904,-45.552,178.889,6.094,149.425
C04160=1139.057,-78.155,-45.541,178.886,6.094,149.426
C04161=1139.063,-78.404,-45.531,178.884,6.093,149.426
C04162=1139.068,-78.653,-45.522,178.882,6.093,149.427
C04163=1139.074,-78.904,-45.512,178.880,6.092,149.427
C04164=1139.079,-79.153,-45.502,178.878,6.092,149.428
C04165=1139.084,-79.402,-45.492,178.875,6.091,149.428
C04166=1139.089,-79.653,-45.482,178.874,6.091,149.429
C04167=1139.095,-79.903,-45.472,178.872,6.090,149.429
C04168=1139.100,-80.152,-45.463,178.869,6.090,149.430
C04169=1139.106,-80.402,-45.453,178.867,6.090,149.430
C04170=1139.111,-80.652,-45.443,178.865,6.089,149.431
C04171=1139.116,-80.901,-45.433,178.863,6.089,149.431
C04172=1139.122,-81.152,-45.423,178.861,6.088,149.432
C04173=1139.126,-81.401,-45.414,178.859,6.088,149.432
C04174=1139.132,-81.651,-45.404,178.856,6.087,149.433
C04175=1139.138,-81.901,-45.394,178.854,6.087,149.434
C04176=1139.143,-82.150,-45.385,178.852,6.086,149.434
C04177=1139.148,-82.399,-45.374,178.850,6.086,149.434
C04178=1139.153,-82.650,-45.365,178.848,6.085,149.435
C04179=1139.159,-82.900,-45.355,178.846,6.085,149.436
C04180=1139.164,-83.150,-45.345,178.843,6.084,149.436
C04181=1139.169,-83.399,-45.336,178.842,6.084,149.437
C04182=1139.175,-83.649,-45.326,178.840,6.083,149.437
C04183=1139.180,-83.898,-45.317,178.837,6.083,149.438
C04184=1139.186,-84.148,-45.306,178.835,6.083,149.438
C04185=1139.191,-84.398,-45.298,178.833,6.082,149.439
C04186=1139.196,-84.648,-45.287,178.831,6.082,149.439
C04187=1139.201,-84.897,-45.277,178.829,6.081,149.440
C04188=1139.207,-85.147,-45.268,178.827,6.081,149.440
C04189=1139.212,-85.397,-45.258,178.824,6.080,149.441
C04190=1139.217,-85.647,-45.249,178.822,6.080,149.441
C04191=1139.223,-85.896,-45.239,178.821,6.080,149.442
C04192=1139.228,-86.146,-45.230,178.819,6.079,149.442
C04193=1139.234,-86.396,-45.219,178.816,6.078,149.443
C04194=1139.239,-86.646,-45.211,178.815,6.078,149.443
C04195=1139.244,-86.896,-45.200,178.812,6.078,149.444
C04196=1139.249,-87.146,-45.191,178.810,6.077,149.445
C04197=1139.255,-87.395,-45.181,178.808,6.076,149.445
C04198=1139.260,-87.645,-45.172,178.806,6.076,149.446
C04199=1139.265,-87.894,-45.162,178.804,6.076,149.446
C04200=1139.271,-88.144,-45.153,178.801,6.075,149.447
C04201=1139.275,-88.394,-45.143,178.800,6.075,149.447
C04202=1139.281,-88.644,-45.134,178.797,6.075,149.448
C04203=1139.287,-88.894,-45.125,178.795,6.074,149.448
C04204=1139.292,-89.143,-45.115,178.794,6.074,149.449
C04205=1139.297,-89.393,-45.106,178.791,6.073,149.449
C04206=1139.303,-89.643,-45.096,178.789,6.073,149.450
C04207=1139.308,-89.892,-45.087,178.787,6.072,149.450
C04208=1139.314,-90.142,-45.076,178.785,6.072,149.451
C04209=1139.319,-90.392,-45.068,178.783,6.071,149.451
C04210=1139.324,-90.642,-45.059,178.781,6.070,149.452
C04211=1139.329,-90.892,-45.048,178.779,6.070,149.452
C04212=1139.334,-91.142,-45.039,178.776,6.070,149.453
C04213=1139.340,-91.391,-45.029,178.774,6.069,149.453
C04214=1139.345,-91.641,-45.020,178.773,6.069,149.454
C04215=1139.350,-91.891,-45.011,178.770,6.069,149.454
C04216=1139.356,-92.141,-45.001,178.768,6.068,149.455
C04217=1139.361,-92.390,-44.992,178.767,6.068,149.455
C04218=1139.367,-92.641,-44.983,178.764,6.068,149.456
C04219=1139.372,-92.890,-44.973,178.762,6.067,149.457
C04220=1139.377,-93.140,-44.964,178.760,6.067,149.457
C04221=1139.383,-93.390,-44.955,178.758,6.066,149.458
C04222=1139.388,-93.639,-44.945,178.756,6.065,149.458
C04223=1139.393,-93.889,-44.935,178.754,6.065,149.459
C04224=1139.399,-94.139,-44.927,178.752,6.065,149.459
C04225=1139.403,-94.388,-44.917,178.749,6.064,149.460
C04226=1139.409,-94.639,-44.907,178.748,6.064,149.460
C04227=1139.415,-94.888,-44.899,178.745,6.064,149.461
C04228=1139.420,-95.138,-44.890,178.743,6.063,149.461
C04229=1139.425,-95.388,-44.879,178.742,6.063,149.462
C04230=1139.431,-95.637,-44.871,178.739,6.062,149.462
C04231=1139.436,-95.887,-44.862,178.737,6.061,149.463
C04232=1139.442,-96.137,-44.853,178.735,6.062,149.463
C04233=1139.447,-96.386,-44.843,178.733,6.061,149.464
C04234=1139.452,-96.636,-44.834,178.731,6.060,149.464
C04235=1139.458,-96.886,-44.825,178.729,6.060,149.465
C04236=1139.463,-97.136,-44.816,178.727,6.059,149.465
C04237=1139.468,-97.385,-44.806,178.725,6.059,149.466
C04238=1139.473,-97.635,-44.797,178.723,6.059,149.466
C04239=1139.479,-97.885,-44.788,178.721,6.058,149.467
C04240=1139.484,-98.135,-44.779,178.719,6.058,149.467
C04241=1139.489,-98.385,-44.770,178.717,6.058,149.468
C04242=1139.495,-98.635,-44.760,178.715,6.057,149.468
C04243=1139.500,-98.884,-44.751,178.713,6.057,149.469
C04244=1139.505,-99.134,-44.742,178.711,6.056,149.469
C04245=1139.511,-99.384,-44.733,178.709,6.055,149.470
C04246=1139.517,-99.634,-44.724,178.707,6.056,149.470
C04247=1139.522,-99.883,-44.715,178.704,6.055,149.471
C04248=1139.527,-100.133,-44.706,178.702,6.054,149.472
C04249=1139.532,-100.382,-44.696,178.700,6.054,149.472
C04250=1139.538,-100.633,-44.687,178.698,6.054,149.473
C04251=1139.543,-100.882,-44.678,178.697,6.054,149.473
C04252=1139.549,-101.132,-44.669,178.694,6.053,149.474
C04253=1139.554,-101.382,-44.660,178.692,6.052,149.474
C04254=1139.560,-101.632,-44.651,178.691,6.052,149.474
C04255=1139.565,-101.882,-44.642,178.688,6.052,149.475
C04256=1139.571,-102.131,-44.633,178.686,6.051,149.476
C04257=1139.576,-102.381,-44.624,178.684,6.051,149.476
C04258=1139.581,-102.653,-44.614,178.682,6.050,149.477
C04259=1139.587,-102.926,-44.605,178.680,6.050,149.477
C04260=1139.592,-103.198,-44.594,178.677,6.049,149.478
C04261=1139.599,-103.470,-44.584,178.676,6.049,149.478
C04262=1139.604,-103.720,-44.575,178.673,6.049,149.479
C04263=1139.610,-103.969,-44.567,178.671,6.048,149.479
C04264=1139.615,-104.219,-44.558,178.670,6.048,149.480
C04265=1139.620,-104.469,-44.549,178.667,6.047,149.480
C04266=1139.625,-104.719,-44.540,178.666,6.047,149.481
C04267=1139.631,-104.969,-44.531,178.663,6.047,149.482
C04268=1139.637,-105.219,-44.522,178.661,6.046,149.482
C04269=1139.642,-105.469,-44.513,178.659,6.046,149.482
C04270=1139.647,-105.718,-44.504,178.657,6.045,149.483
C04271=1139.653,-105.968,-44.495,178.656,6.045,149.483
C04272=1139.658,-106.218,-44.487,178.653,6.045,149.484
C04273=1139.663,-106.468,-44.478,178.651,6.044,149.484
C04274=1139.668,-106.717,-44.469,178.650,6.044,149.485
C04275=1139.673,-106.967,-44.460,178.647,6.043,149.485
C04276=1139.680,-107.217,-44.451,178.646,6.043,149.486
C04277=1139.685,-107.467,-44.442,178.643,6.043,149.487
C04278=1139.690,-107.716,-44.433,178.641,6.042,149.487
C04279=1139.695,-107.966,-44.424,178.639,6.042,149.488
C04280=1139.700,-108.216,-44.415,178.637,6.041,149.488
C04281=1139.706,-108.465,-44.407,178.635,6.041,149.489
C04282=1139.711,-108.715,-44.398,178.633,6.041,149.489
C04283=1139.717,-108.965,-44.389,178.631,6.040,149.490
C04284=1139.722,-109.215,-44.380,178.629,6.040,149.490
C04285=1139.727,-109.465,-44.371,178.627,6.039,149.490
C04286=1139.733,-109.714,-44.363,178.626,6.039,149.491
C04287=1139.738,-109.964,-44.354,178.623,6.039,149.491
C04288=1139.744,-110.214,-44.345,178.621,6.038,149.492
C04289=1139.749,-110.464,-44.336,178.620,6.038,149.492
C04290=1139.754,-110.714,-44.327,178.617,6.038,149.493
C04291=1139.760,-110.963,-44.318,178.615,6.038,149.494
C04292=1139.765,-111.213,-44.310,178.613,6.037,149.494
C04293=1139.770,-111.463,-44.301,178.612,6.037,149.495
C04294=1139.776,-111.714,-44.293,178.609,6.036,149.495
C04295=1139.782,-111.963,-44.284,178.607,6.035,149.496
C04296=1139.787,-112.213,-44.275,178.606,6.035,149.496
C04297=1139.792,-112.462,-44.266,178.603,6.035,149.497
C04298=1139.797,-112.712,-44.257,178.602,6.035,149.497
C04299=1139.803,-112.961,-44.249,178.600,6.034,149.498
C04300=1139.808,-113.212,-44.241,178.597,6.033,149.498
C04301=1139.814,-113.462,-44.232,178.596,6.033,149.499
C04302=1139.819,-113.712,-44.223,178.594,6.032,149.499
C04303=1139.825,-113.961,-44.214,178.592,6.033,149.499
C04304=1139.830,-114.211,-44.206,178.590,6.032,149.500
C04305=1139.835,-114.461,-44.197,178.588,6.032,149.500
C04306=1139.840,-114.711,-44.188,178.586,6.031,149.501
C04307=1139.846,-114.960,-44.180,178.584,6.032,149.502
C04308=1139.851,-115.210,-44.171,178.582,6.031,149.502
C04309=1139.857,-115.460,-44.163,178.580,6.030,149.503
C04310=1139.863,-115.709,-44.154,178.578,6.030,149.503
C04311=1139.868,-115.959,-44.145,178.576,6.029,149.504
C04312=1139.873,-116.210,-44.137,178.574,6.029,149.504
C04313=1139.879,-116.459,-44.129,178.572,6.029,149.505
C04314=1139.883,-116.708,-44.120,178.570,6.029,149.505
C04315=1139.889,-116.958,-44.111,178.568,6.028,149.506
C04316=1139.894,-117.209,-44.103,178.566,6.027,149.506
C04317=1139.900,-117.458,-44.095,178.564,6.027,149.507
C04318=1139.905,-117.708,-44.086,178.562,6.026,149.507
C04319=1139.910,-117.958,-44.078,178.561,6.027,149.508
C04320=1139.916,-118.207,-44.069,178.558,6.026,149.508
C04321=1139.921,-118.457,-44.060,178.557,6.026,149.508
C04322=1139.927,-118.708,-44.052,178.555,6.025,149.509
C04323=1139.933,-118.957,-44.043,178.553,6.025,149.509
C04324=1139.938,-119.207,-44.034,178.551,6.024,149.510
C04325=1139.942,-119.457,-44.027,178.549,6.024,149.510
C04326=1139.948,-119.706,-44.018,178.547,6.024,149.511
C04327=1139.953,-119.956,-44.009,178.545,6.023,149.511
C04328=1139.959,-120.206,-44.001,178.543,6.023,149.512
C04329=1139.965,-120.456,-43.993,178.541,6.022,149.512
C04330=1139.970,-120.705,-43.984,178.539,6.022,149.513
C04331=1139.975,-120.956,-43.976,178.537,6.022,149.513
C04332=1139.981,-121.205,-43.967,178.536,6.022,149.514
C04333=1139.986,-121.455,-43.960,178.533,6.021,149.514
C04334=1139.991,-121.705,-43.951,178.532,6.021,149.515
C04335=1139.997,-121.954,-43.942,178.530,6.020,149.515
C04336=1140.002,-122.205,-43.934,178.528,6.020,149.516
C04337=1140.008,-122.454,-43.925,178.526,6.019,149.516
C04338=1140.013,-122.704,-43.917,178.524,6.019,149.517
C04339=1140.018,-122.954,-43.909,178.522,6.019,149.517
C04340=1140.024,-123.204,-43.901,178.521,6.019,149.518
C04341=1140.029,-123.453,-43.892,178.518,6.018,149.518
C04342=1140.035,-123.704,-43.884,178.516,6.017,149.519
C04343=1140.040,-123.953,-43.875,178.515,6.017,149.519
C04344=1140.045,-124.203,-43.867,178.512,6.017,149.520
C04345=1140.051,-124.452,-43.859,178.511,6.017,149.520
C04346=1140.056,-124.702,-43.850,178.509,6.016,149.521
C04347=1140.061,-124.953,-43.842,178.507,6.016,149.521
C04348=1140.067,-125.202,-43.834,178.505,6.015,149.522
C04349=1140.072,-125.452,-43.826,178.503,6.015,149.522
C04350=1140.078,-125.701,-43.818,178.501,6.014,149.523
C04351=1140.083,-125.952,-43.809,178.499,6.015,149.523
C04352=1140.089,-126.201,-43.801,178.497,6.014,149.524
C04353=1140.094,-126.451,-43.793,178.496,6.014,149.524
C04354=1140.099,-126.701,-43.784,178.493,6.013,149.525
C04355=1140.105,-126.951,-43.777,178.492,6.013,149.525
C04356=1140.110,-127.201,-43.768,178.490,6.012,149.526
C04357=1140.115,-127.450,-43.760,178.488,6.012,149.526
C04358=1140.121,-127.700,-43.752,178.486,6.012,149.527
C04359=1140.127,-127.949,-43.744,178.484,6.012,149.527
C04360=1140.132,-128.200,-43.736,178.482,6.011,149.528
C04361=1140.137,-128.449,-43.727,178.480,6.011,149.528
C04362=1139.716,-128.461,-43.771,178.477,6.014,149.530
C04363=1139.711,-128.210,-43.779,178.479,6.015,149.529
C04364=1139.705,-127.961,-43.788,178.480,6.015,149.529
C04365=1139.700,-127.711,-43.795,178.483,6.016,149.528
C04366=1139.695,-127.462,-43.804,178.484,6.016,149.528
C04367=1139.689,-127.211,-43.812,178.486,6.016,149.527
C04368=1139.684,-126.962,-43.821,178.488,6.016,149.527
C04369=1139.679,-126.712,-43.828,178.490,6.017,149.526
C04370=1139.673,-126.462,-43.837,178.492,6.017,149.526
C04371=1139.667,-126.213,-43.845,178.494,6.018,149.525
C04372=1139.662,-125.963,-43.854,178.495,6.018,149.525
C04373=1139.657,-125.713,-43.861,178.498,6.019,149.524
C04374=1139.652,-125.463,-43.870,178.499,6.019,149.524
C04375=1139.646,-125.213,-43.878,178.501,6.019,149.523
C04376=1139.640,-124.964,-43.886,178.503,6.019,149.523
C04377=1139.635,-124.713,-43.895,178.505,6.020,149.522
C04378=1139.630,-124.464,-43.903,178.507,6.020,149.522
C04379=1139.624,-124.214,-43.911,178.509,6.021,149.522
C04380=1139.619,-123.964,-43.920,178.511,6.021,149.521
C04381=1139.613,-123.714,-43.927,178.513,6.021,149.521
C04382=1139.608,-123.465,-43.936,178.515,6.022,149.520
C04383=1139.603,-123.215,-43.944,178.517,6.022,149.520
C04384=1139.598,-122.965,-43.952,178.519,6.023,149.519
C04385=1139.592,-122.715,-43.961,178.520,6.023,149.519
C04386=1139.586,-122.466,-43.969,178.523,6.023,149.518
C04387=1139.581,-122.215,-43.977,178.524,6.023,149.518
C04388=1139.576,-121.966,-43.986,178.526,6.024,149.517
C04389=1139.571,-121.716,-43.994,178.528,6.024,149.517
C04390=1139.565,-121.466,-44.002,178.530,6.025,149.516
C04391=1139.560,-121.216,-44.011,178.532,6.025,149.516
C04392=1139.554,-120.966,-44.019,178.534,6.026,149.515
C04393=1139.549,-120.716,-44.028,178.536,6.026,149.515
C04394=1139.543,-120.467,-44.037,178.538,6.026,149.514
C04395=1139.538,-120.217,-44.044,178.539,6.026,149.514
C04396=1139.533,-119.967,-44.053,178.542,6.027,149.513
C04397=1139.527,-119.718,-44.062,178.544,6.028,149.513
C04398=1139.522,-119.468,-44.070,178.545,6.028,149.512
C04399=1139.517,-119.218,-44.079,178.548,6.028,149.512
C04400=1139.511,-118.968,-44.086,178.549,6.028,149.511
C04401=1139.505,-118.718,-44.095,178.551,6.029,149.511
C04402=1139.500,-118.468,-44.104,178.553,6.029,149.510
C04403=1139.495,-118.219,-44.111,178.555,6.030,149.510
C04404=1139.490,-117.969,-44.120,178.557,6.030,149.509
C04405=1139.485,-117.719,-44.129,178.559,6.031,149.509
C04406=1139.479,-117.469,-44.137,178.561,6.030,149.508
C04407=1139.473,-117.220,-44.146,178.563,6.031,149.508
C04408=1139.468,-116.970,-44.155,178.565,6.032,149.507
C04409=1139.463,-116.720,-44.164,178.567,6.032,149.507
C04410=1139.457,-116.470,-44.172,178.569,6.033,149.506
C04411=1139.452,-116.220,-44.180,178.570,6.033,149.506
C04412=1139.447,-115.970,-44.189,178.573,6.033,149.505
C04413=1139.441,-115.721,-44.197,178.574,6.033,149.505
C04414=1139.435,-115.471,-44.206,178.576,6.034,149.504
C04415=1139.430,-115.221,-44.215,178.578,6.034,149.504
C04416=1139.424,-114.972,-44.223,178.581,6.034,149.503
C04417=1139.419,-114.721,-44.232,178.583,6.035,149.503
C04418=1139.414,-114.471,-44.241,178.584,6.035,149.502
C04419=1139.409,-114.222,-44.249,178.587,6.036,149.502
C04420=1139.403,-113.973,-44.258,178.588,6.036,149.501
C04421=1139.398,-113.723,-44.267,178.590,6.037,149.501
C04422=1139.392,-113.472,-44.275,178.592,6.037,149.500
C04423=1139.387,-113.222,-44.284,178.594,6.037,149.500
C04424=1139.381,-112.973,-44.293,178.596,6.038,149.499
C04425=1139.376,-112.723,-44.301,178.598,6.038,149.499
C04426=1139.371,-112.473,-44.310,178.600,6.039,149.498
C04427=1139.365,-112.223,-44.318,178.602,6.039,149.498
C04428=1139.360,-111.974,-44.327,178.604,6.039,149.497
C04429=1139.355,-111.724,-44.336,178.606,6.039,149.497
C04430=1139.349,-111.474,-44.345,178.608,6.040,149.496
C04431=1139.344,-111.224,-44.354,178.610,6.041,149.496
C04432=1139.338,-110.975,-44.362,178.612,6.041,149.495
C04433=1139.333,-110.725,-44.370,178.614,6.042,149.495
C04434=1139.328,-110.475,-44.379,178.616,6.041,149.494
C04435=1139.323,-110.225,-44.388,178.618,6.042,149.494
C04436=1139.317,-109.976,-44.397,178.620,6.043,149.493
C04437=1139.312,-109.726,-44.406,178.622,6.043,149.493
C04438=1139.307,-109.476,-44.415,178.624,6.043,149.492
C04439=1139.301,-109.226,-44.423,178.626,6.043,149.492
C04440=1139.296,-108.976,-44.432,178.628,6.044,149.491
C04441=1139.290,-108.727,-44.441,178.630,6.045,149.491
C04442=1139.285,-108.477,-44.449,178.632,6.045,149.490
C04443=1139.280,-108.227,-44.458,178.634,6.046,149.490
C04444=1139.275,-107.977,-44.467,178.635,6.045,149.489
C04445=1139.269,-107.727,-44.476,178.638,6.046,149.489
C04446=1139.263,-107.478,-44.485,178.639,6.046,149.488
C04447=1139.258,-107.228,-44.494,178.642,6.047,149.488
C04448=1139.253,-106.978,-44.503,178.644,6.047,149.487
C04449=1139.247,-106.728,-44.512,178.646,6.047,149.487
C04450=1139.242,-106.478,-44.520,178.648,6.048,149.486
C04451=1139.237,-106.229,-44.529,178.650,6.049,149.486
C04452=1139.231,-105.979,-44.538,178.652,6.049,149.485
C04453=1139.226,-105.730,-44.547,178.654,6.049,149.485
C04454=1139.220,-105.479,-44.556,178.655,6.049,149.484
C04455=1139.215,-105.230,-44.565,178.658,6.050,149.484
C04456=1139.210,-104.980,-44.574,178.660,6.051,149.483
C04457=1139.205,-104.730,-44.583,178.661,6.051,149.483
C04458=1139.199,-104.481,-44.592,178.664,6.051,149.482
C04459=1139.194,-104.231,-44.600,178.666,6.051,149.482
C04460=1139.189,-103.981,-44.609,178.668,6.052,149.481
C04461=1139.183,-103.731,-44.619,178.670,6.053,149.481
C04462=1139.178,-103.481,-44.628,178.672,6.053,149.480
C04463=1139.172,-103.209,-44.638,178.674,6.053,149.480
C04464=1139.166,-102.936,-44.647,178.677,6.054,149.479
C04465=1139.160,-102.665,-44.657,178.679,6.054,149.478
C04466=1139.154,-102.393,-44.667,178.680,6.054,149.478
C04467=1139.149,-102.143,-44.676,178.683,6.055,149.478
C04468=1139.144,-101.893,-44.685,178.685,6.056,149.477
C04469=1139.138,-101.643,-44.694,178.686,6.056,149.477
C04470=1139.133,-101.393,-44.703,178.689,6.056,149.476
C04471=1139.128,-101.143,-44.712,178.691,6.056,149.475
C04472=1139.123,-100.893,-44.721,178.693,6.057,149.475
C04473=1139.117,-100.644,-44.731,178.695,6.058,149.474
C04474=1139.111,-100.395,-44.740,178.697,6.058,149.474
C04475=1139.106,-100.145,-44.748,178.699,6.058,149.473
C04476=1139.101,-99.895,-44.757,178.701,6.059,149.473
C04477=1139.095,-99.645,-44.767,178.703,6.059,149.472
C04478=1139.090,-99.395,-44.776,178.705,6.060,149.472
C04479=1139.085,-99.145,-44.785,178.708,6.060,149.471
C04480=1139.080,-98.896,-44.794,178.709,6.060,149.471
C04481=1139.074,-98.646,-44.804,178.711,6.061,149.470
C04482=1139.069,-98.396,-44.813,178.713,6.061,149.470
C04483=1139.064,-98.146,-44.822,178.715,6.062,149.469
C04484=1139.059,-97.896,-44.830,178.717,6.062,149.469
C04485=1139.052,-97.647,-44.840,178.719,6.062,149.468
C04486=1139.047,-97.397,-44.849,178.721,6.063,149.468
C04487=1139.042,-97.148,-44.858,178.724,6.064,149.467
C04488=1139.036,-96.897,-44.868,178.725,6.064,149.467
C04489=1139.031,-96.648,-44.876,178.728,6.064,149.466
C04490=1139.026,-96.398,-44.886,178.730,6.065,149.466
C04491=1139.020,-96.148,-44.896,178.731,6.065,149.465
C04492=1139.015,-95.898,-44.904,178.734,6.066,149.465
C04493=1139.010,-95.648,-44.913,178.736,6.066,149.464
C04494=1139.004,-95.399,-44.924,178.738,6.066,149.464
C04495=1138.999,-95.149,-44.932,178.740,6.067,149.463
C04496=1138.994,-94.899,-44.941,178.742,6.068,149.463
C04497=1138.988,-94.649,-44.951,178.744,6.068,149.462
C04498=1138.983,-94.400,-44.960,178.746,6.068,149.462
C04499=1138.978,-94.150,-44.969,178.748,6.069,149.461
C04500=1138.972,-93.900,-44.979,178.750,6.069,149.461
C04501=1138.967,-93.651,-44.988,178.752,6.069,149.460
C04502=1138.962,-93.401,-44.997,178.755,6.070,149.459
C04503=1138.956,-93.151,-45.007,178.756,6.070,149.459
C04504=1138.951,-92.901,-45.016,178.758,6.071,149.458
C04505=1138.945,-92.651,-45.026,178.761,6.072,149.458
C04506=1138.940,-92.401,-45.035,178.762,6.072,149.457
C04507=1138.935,-92.151,-45.044,178.764,6.072,149.457
C04508=1138.929,-91.902,-45.054,178.767,6.073,149.456
C04509=1138.924,-91.652,-45.063,178.769,6.073,149.456
C04510=1138.919,-91.403,-45.072,178.771,6.073,149.455
C04511=1138.913,-91.153,-45.082,178.773,6.074,149.455
C04512=1138.908,-90.903,-45.091,178.775,6.074,149.454
C04513=1138.903,-90.653,-45.101,178.777,6.075,149.454
C04514=1138.898,-90.403,-45.110,178.780,6.075,149.453
C04515=1138.892,-90.153,-45.119,178.781,6.075,149.453
C04516=1138.887,-89.904,-45.129,178.783,6.076,149.452
C04517=1138.882,-89.654,-45.138,178.786,6.077,149.452
C04518=1138.876,-89.405,-45.148,178.787,6.077,149.451
C04519=1138.871,-89.155,-45.157,178.789,6.077,149.451
C04520=1138.865,-88.905,-45.167,178.792,6.078,149.450
C04521=1138.860,-88.655,-45.176,178.794,6.079,149.450
C04522=1138.854,-88.405,-45.186,178.796,6.079,149.449
C04523=1138.850,-88.155,-45.196,178.798,6.079,149.449
C04524=1138.844,-87.905,-45.205,178.800,6.080,149.448
C04525=1138.839,-87.656,-45.215,178.802,6.080,149.448
C04526=1138.833,-87.406,-45.224,178.804,6.080,149.447
C04527=1138.828,-87.156,-45.234,178.807,6.081,149.446
C04528=1138.823,-86.906,-45.243,178.808,6.081,149.446
C04529=1138.818,-86.657,-45.253,178.810,6.082,149.445
C04530=1138.812,-86.407,-45.262,178.813,6.083,149.445
C04531=1138.807,-86.158,-45.272,178.815,6.083,149.444
C04532=1138.801,-85.908,-45.282,178.817,6.083,149.444
C04533=1138.796,-85.658,-45.291,178.819,6.084,149.443
C04534=1138.791,-85.407,-45.301,178.821,6.084,149.443
C04535=1138.786,-85.158,-45.311,178.823,6.084,149.442
C04536=1138.780,-84.908,-45.320,178.825,6.085,149.442
C04537=1138.775,-84.659,-45.330,178.828,6.086,149.441
C04538=1138.770,-84.409,-45.340,178.830,6.086,149.441
C04539=1138.764,-84.159,-45.349,178.832,6.086,149.440
C04540=1138.759,-83.910,-45.359,178.834,6.087,149.440
C04541=1138.754,-83.660,-45.368,178.836,6.088,149.439
C04542=1138.748,-83.410,-45.378,178.838,6.087,149.438
C04543=1138.743,-83.160,-45.387,178.840,6.088,149.438
C04544=1138.738,-82.910,-45.398,178.842,6.089,149.437
C04545=1138.732,-82.661,-45.408,178.845,6.090,149.437
C04546=1138.727,-82.411,-45.417,178.846,6.090,149.437
C04547=1138.722,-82.161,-45.427,178.849,6.090,149.436
C04548=1138.717,-81.912,-45.437,178.851,6.091,149.435
C04549=1138.711,-81.662,-45.446,178.853,6.091,149.435
C04550=1138.706,-81.412,-45.457,178.855,6.091,149.434
C04551=1138.701,-81.162,-45.466,178.857,6.092,149.434
C04552=1138.695,-80.912,-45.476,178.860,6.093,149.433
C04553=1138.690,-80.663,-45.485,178.861,6.093,149.433
C04554=1138.684,-80.413,-45.495,178.863,6.093,149.432
C04555=1138.679,-80.163,-45.505,178.866,6.094,149.432
C04556=1138.674,-79.914,-45.515,178.868,6.095,149.431
C04557=1138.668,-79.663,-45.525,178.870,6.094,149.431
C04558=1138.663,-79.414,-45.535,178.872,6.095,149.430
C04559=1138.658,-79.165,-45.544,178.874,6.096,149.430
C04560=1138.652,-78.915,-45.555,178.877,6.097,149.429
C04561=1138.647,-78.665,-45.564,178.878,6.097,149.429
C04562=1138.642,-78.415,-45.574,178.881,6.097,149.428
C04563=1138.637,-78.165,-45.584,178.883,6.098,149.427
C04564=1138.631,-77.915,-45.594,178.885,6.099,149.427
C04565=1138.626,-77.666,-45.603,178.887,6.099,149.426
C04566=1138.620,-77.416,-45.614,178.889,6.099,149.426
C04567=1138.615,-77.145,-45.625,178.892,6.100,149.425
C04568=1138.609,-76.873,-45.635,178.894,6.100,149.425
C04569=1138.604,-76.602,-45.646,178.896,6.101,149.424
C04570=1138.597,-76.330,-45.657,178.899,6.102,149.424
C04571=1138.592,-76.081,-45.666,178.900,6.102,149.423
C04572=1138.587,-75.831,-45.677,178.903,6.102,149.422
C04573=1138.581,-75.581,-45.687,178.905,6.103,149.422
C04574=1138.576,-75.332,-45.697,178.907,6.103,149.421
C04575=1138.571,-75.082,-45.706,178.910,6.104,149.421
C04576=1138.566,-74.831,-45.717,178.911,6.104,149.420
C04577=1138.560,-74.582,-45.727,178.914,6.105,149.420
C04578=1138.554,-74.332,-45.737,178.916,6.105,149.419
C04579=1138.550,-74.083,-45.747,178.918,6.106,149.419
C04580=1138.545,-73.833,-45.757,178.920,6.106,149.418
C04581=1138.539,-73.583,-45.767,178.922,6.106,149.418
C04582=1138.533,-73.333,-45.777,178.925,6.107,149.417
C04583=1138.527,-73.084,-45.787,178.927,6.108,149.417
C04584=1138.523,-72.834,-45.797,178.928,6.108,149.416
C04585=1138.518,-72.584,-45.808,178.931,6.109,149.416
C04586=1138.512,-72.335,-45.818,178.933,6.109,149.415
C04587=1138.506,-72.085,-45.828,178.935,6.110,149.414
C04588=1138.502,-71.835,-45.838,178.938,6.111,149.414
C04589=1138.496,-71.585,-45.847,178.939,6.111,149.413
C04590=1138.491,-71.335,-45.858,178.942,6.111,149.413
C04591=1138.486,-71.085,-45.868,178.944,6.112,149.412
C04592=1138.480,-70.836,-45.878,178.946,6.112,149.412
C04593=1138.474,-70.586,-45.889,178.948,6.112,149.411
C04594=1138.470,-70.336,-45.899,178.951,6.113,149.411
C04595=1138.465,-70.087,-45.909,178.953,6.114,149.410
C04596=1138.459,-69.837,-45.919,178.955,6.114,149.410
C04597=1138.453,-69.588,-45.929,178.957,6.115,149.409
C04598=1138.448,-69.337,-45.940,178.959,6.115,149.408
C04599=1138.443,-69.088,-45.950,178.961,6.115,149.408
C04600=1138.437,-68.838,-45.960,178.964,6.116,149.408
C04601=1138.433,-68.588,-45.970,178.966,6.117,149.407
C04602=1138.427,-68.339,-45.980,178.968,6.117,149.406
C04603=1138.422,-68.089,-45.991,178.970,6.117,149.406
C04604=1138.417,-67.839,-46.001,178.972,6.118,149.405
C04605=1138.411,-67.589,-46.011,178.974,6.119,149.405
C04606=1138.406,-67.340,-46.022,178.977,6.119,149.404
C04607=1138.401,-67.090,-46.032,178.979,6.120,149.404
C04608=1138.395,-66.840,-46.042,178.981,6.120,149.403
C04609=1138.390,-66.590,-46.053,178.983,6.121,149.403
C04610=1138.385,-66.341,-46.063,178.986,6.121,149.402
C04611=1138.380,-66.091,-46.073,178.988,6.122,149.402
C04612=1138.375,-65.841,-46.084,178.990,6.123,149.401
C04613=1138.369,-65.592,-46.094,178.992,6.123,149.401
C04614=1138.364,-65.342,-46.105,178.994,6.123,149.400
C04615=1138.359,-65.092,-46.115,178.997,6.124,149.399
C04616=1138.353,-64.843,-46.125,178.999,6.125,149.399
C04617=1138.348,-64.592,-46.136,179.001,6.125,149.398
C04618=1138.342,-64.343,-46.146,179.004,6.126,149.398
C04619=1138.337,-64.093,-46.156,179.005,6.126,149.397
C04620=1138.332,-63.843,-46.167,179.007,6.126,149.397
C04621=1138.327,-63.594,-46.178,179.010,6.127,149.396
C04622=1138.322,-63.344,-46.188,179.012,6.128,149.396
C04623=1138.316,-63.094,-46.199,179.014,6.128,149.395
C04624=1138.310,-62.845,-46.209,179.017,6.129,149.395
C04625=1138.305,-62.594,-46.219,179.018,6.129,149.394
C04626=1138.300,-62.345,-46.230,179.021,6.129,149.393
C04627=1138.295,-62.095,-46.241,179.023,6.130,149.393
C04628=1138.289,-61.846,-46.251,179.025,6.131,149.392
C04629=1138.284,-61.596,-46.262,179.028,6.132,149.392
C04630=1138.279,-61.346,-46.272,179.030,6.132,149.391
C04631=1138.273,-61.096,-46.282,179.032,6.132,149.391
C04632=1138.269,-60.847,-46.293,179.034,6.133,149.390
C04633=1138.263,-60.597,-46.304,179.037,6.133,149.390
C04634=1138.258,-60.347,-46.314,179.039,6.134,149.389
C04635=1138.252,-60.097,-46.324,179.041,6.135,149.389
C04636=1138.248,-59.848,-46.336,179.043,6.136,149.388
C04637=1138.242,-59.598,-46.346,179.046,6.136,149.387
C04638=1138.237,-59.348,-46.356,179.047,6.136,149.387
C04639=1138.232,-59.099,-46.367,179.050,6.137,149.387
C04640=1138.227,-58.849,-46.378,179.052,6.138,149.386
C04641=1138.221,-58.599,-46.388,179.055,6.138,149.385
C04642=1138.216,-58.349,-46.399,179.057,6.139,149.385
C04643=1138.211,-58.100,-46.410,179.059,6.139,149.384
C04644=1138.206,-57.850,-46.420,179.062,6.140,149.384
C04645=1138.200,-57.600,-46.430,179.063,6.140,149.383
C04646=1138.195,-57.350,-46.442,179.065,6.141,149.383
C04647=1138.189,-57.101,-46.452,179.068,6.141,149.382
C04648=1138.184,-56.851,-46.463,179.070,6.142,149.382
C04649=1138.179,-56.602,-46.474,179.072,6.142,149.381
C04650=1138.174,-56.352,-46.485,179.075,6.143,149.381
C04651=1138.168,-56.102,-46.495,179.077,6.144,149.380
C04652=1138.164,-55.852,-46.506,179.079,6.144,149.379
C04653=1138.158,-55.603,-46.516,179.081,6.144,149.379
C04654=1138.153,-55.353,-46.528,179.083,6.145,149.378
C04655=1138.147,-55.103,-46.538,179.086,6.146,149.378
C04656=1138.142,-54.853,-46.549,179.088,6.146,149.377
C04657=1138.137,-54.604,-46.560,179.090,6.147,149.377
C04658=1138.132,-54.354,-46.570,179.093,6.147,149.376
C04659=1138.127,-54.105,-46.581,179.095,6.148,149.376
C04660=1138.122,-53.855,-46.592,179.097,6.149,149.375
C04661=1138.115,-53.606,-46.603,179.099,6.149,149.375
C04662=1138.110,-53.355,-46.614,179.102,6.149,149.374
C04663=1138.105,-53.105,-46.625,179.104,6.150,149.373
C04664=1138.100,-52.856,-46.636,179.106,6.151,149.373
C04665=1138.095,-52.606,-46.646,179.109,6.151,149.372
C04666=1138.089,-52.357,-46.658,179.111,6.152,149.372
C04667=1138.084,-52.106,-46.668,179.113,6.153,149.371
C04668=1138.079,-51.857,-46.679,179.115,6.154,149.371
C04669=1138.074,-51.607,-46.690,179.118,6.154,149.370
C04670=1138.069,-51.358,-46.701,179.119,6.154,149.370
C04671=1138.063,-51.087,-46.713,179.122,6.154,149.369
C04672=1138.057,-50.816,-46.725,179.125,6.156,149.368
C04673=1138.051,-50.545,-46.736,179.128,6.156,149.368
C04674=1138.046,-50.275,-46.748,179.130,6.157,149.367
C04675=1138.041,-50.025,-46.760,179.132,6.158,149.367
C04676=1138.035,-49.775,-46.770,179.134,6.158,149.366
C04677=1138.030,-49.526,-46.781,179.136,6.158,149.366
C04678=1138.024,-49.276,-46.793,179.138,6.159,149.365
C04679=1138.019,-49.026,-46.803,179.141,6.159,149.364
C04680=1138.015,-48.777,-46.815,179.143,6.160,149.364
C04681=1138.009,-48.527,-46.825,179.145,6.161,149.363
C04682=1138.003,-48.277,-46.837,179.148,6.162,149.363
C04683=1137.999,-48.027,-46.848,179.150,6.162,149.362
C04684=1137.993,-47.778,-46.858,179.153,6.163,149.362
C04685=1137.988,-47.528,-46.870,179.155,6.164,149.361
C04686=1137.982,-47.278,-46.880,179.157,6.164,149.361
C04687=1137.977,-47.029,-46.892,179.160,6.165,149.360
C04688=1137.972,-46.779,-46.904,179.161,6.165,149.360
C04689=1137.966,-46.529,-46.914,179.164,6.165,149.359
C04690=1137.962,-46.280,-46.925,179.166,6.166,149.358
C04691=1137.956,-46.030,-46.937,179.168,6.167,149.358
C04692=1137.951,-45.780,-46.947,179.170,6.168,149.358
C04693=1137.946,-45.531,-46.958,179.173,6.168,149.357
C04694=1137.941,-45.281,-46.970,179.175,6.169,149.356
C04695=1137.935,-45.031,-46.981,179.177,6.170,149.356
C04696=1137.930,-44.781,-46.992,179.180,6.170,149.355
C04697=1137.925,-44.532,-47.004,179.182,6.171,149.355
C04698=1137.920,-44.283,-47.015,179.184,6.171,149.354
C04699=1137.914,-44.032,-47.026,179.187,6.172,149.353
C04700=1137.909,-43.782,-47.037,179.189,6.173,149.353
C04701=1137.904,-43.533,-47.048,179.192,6.173,149.353
C04702=1137.898,-43.284,-47.060,179.194,6.174,149.352
C04703=1137.893,-43.033,-47.070,179.196,6.175,149.351
C04704=1137.888,-42.783,-47.082,179.198,6.175,149.351
C04705=1137.883,-42.534,-47.093,179.201,6.175,149.350
C04706=1137.877,-42.285,-47.105,179.203,6.176,149.350
C04707=1137.873,-42.035,-47.116,179.205,6.177,149.349
C04708=1137.867,-41.785,-47.127,179.208,6.177,149.349
C04709=1137.862,-41.535,-47.139,179.210,6.178,149.348
C04710=1137.857,-41.286,-47.150,179.212,6.178,149.348
C04711=1137.851,-41.036,-47.162,179.214,6.179,149.347
C04712=1137.846,-40.787,-47.173,179.217,6.180,149.346
C04713=1137.840,-40.536,-47.184,179.219,6.180,149.346
C04714=1137.836,-40.287,-47.195,179.221,6.181,149.345
C04715=1137.830,-40.037,-47.207,179.224,6.182,149.345
C04716=1137.825,-39.788,-47.218,179.226,6.182,149.344
C04717=1137.820,-39.538,-47.230,179.228,6.183,149.344
C04718=1137.815,-39.288,-47.241,179.231,6.184,149.343
C04719=1137.809,-39.038,-47.253,179.233,6.184,149.343
C04720=1137.804,-38.789,-47.264,179.235,6.185,149.342
C04721=1137.798,-38.539,-47.275,179.238,6.186,149.341
C04722=1137.794,-38.289,-47.286,179.240,6.186,149.341
C04723=1137.788,-38.039,-47.298,179.242,6.187,149.340
C04724=1137.783,-37.790,-47.309,179.245,6.187,149.340
C04725=1137.778,-37.540,-47.321,179.247,6.188,149.339
C04726=1137.773,-37.291,-47.332,179.249,6.189,149.339
C04727=1137.767,-37.041,-47.344,179.252,6.189,149.338
C04728=1137.762,-36.791,-47.356,179.254,6.190,149.338
C04729=1137.757,-36.542,-47.367,179.256,6.191,149.337
C04730=1137.751,-36.292,-47.379,179.259,6.191,149.336
C04731=1137.747,-36.042,-47.390,179.261,6.192,149.336
C04732=1137.741,-35.793,-47.402,179.264,6.193,149.336
C04733=1137.737,-35.543,-47.413,179.266,6.193,149.335
C04734=1137.730,-35.294,-47.425,179.268,6.194,149.334
C04735=1137.725,-35.044,-47.437,179.271,6.195,149.334
C04736=1137.720,-34.794,-47.448,179.273,6.195,149.333
C04737=1137.715,-34.544,-47.460,179.275,6.196,149.333
C04738=1137.710,-34.295,-47.471,179.278,6.197,149.332
C04739=1137.705,-34.045,-47.483,179.280,6.197,149.332
C04740=1137.699,-33.795,-47.495,179.282,6.198,149.331
C04741=1137.694,-33.546,-47.506,179.285,6.199,149.331
C04742=1137.689,-33.296,-47.518,179.287,6.199,149.330
C04743=1137.683,-33.046,-47.530,179.289,6.200,149.329
C04744=1137.679,-32.796,-47.541,179.292,6.201,149.329
C04745=1137.673,-32.547,-47.554,179.294,6.201,149.328
C04746=1137.669,-32.297,-47.565,179.297,6.202,149.328
C04747=1137.663,-32.048,-47.576,179.299,6.203,149.327
C04748=1137.657,-31.798,-47.588,179.301,6.203,149.327
C04749=1137.653,-31.549,-47.600,179.304,6.204,149.326
C04750=1137.647,-31.299,-47.612,179.306,6.205,149.326
C04751=1137.642,-31.049,-47.623,179.308,6.205,149.325
C04752=1137.637,-30.799,-47.635,179.311,6.206,149.324
C04753=1137.632,-30.550,-47.647,179.313,6.207,149.324
C04754=1137.626,-30.300,-47.659,179.315,6.207,149.323
C04755=1137.621,-30.050,-47.671,179.318,6.208,149.323
C04756=1137.616,-29.801,-47.682,179.320,6.209,149.322
C04757=1137.610,-29.551,-47.694,179.322,6.209,149.322
C04758=1137.605,-29.301,-47.706,179.325,6.210,149.321
C04759=1137.600,-29.052,-47.718,179.327,6.211,149.321
C04760=1137.595,-28.802,-47.730,179.329,6.211,149.320
C04761=1137.590,-28.552,-47.742,179.332,6.212,149.320
C04762=1137.584,-28.302,-47.753,179.334,6.213,149.319
C04763=1137.580,-28.053,-47.765,179.337,6.213,149.318
C04764=1137.574,-27.803,-47.777,179.339,6.214,149.318
C04765=1137.569,-27.553,-47.789,179.341,6.215,149.317
C04766=1137.564,-27.303,-47.801,179.344,6.215,149.317
C04767=1137.559,-27.054,-47.813,179.346,6.216,149.316
C04768=1137.554,-26.804,-47.825,179.348,6.217,149.316
C04769=1137.548,-26.555,-47.837,179.351,6.217,149.315
C04770=1137.543,-26.305,-47.849,179.353,6.218,149.315
C04771=1137.538,-26.055,-47.861,179.355,6.219,149.314
C04772=1137.532,-25.806,-47.872,179.358,6.220,149.313
C04773=1137.527,-25.556,-47.884,179.360,6.221,149.313
C04774=1137.522,-25.307,-47.897,179.363,6.221,149.312
C04775=1137.517,-25.037,-47.910,179.365,6.222,149.312
C04776=1137.511,-24.766,-47.923,179.367,6.223,149.311
C04777=1137.505,-24.497,-47.935,179.370,6.223,149.311
C04778=1137.499,-24.226,-47.949,179.373,6.224,149.310
C04779=1137.495,-23.977,-47.961,179.376,6.225,149.309
C04780=1137.489,-23.727,-47.973,179.378,6.226,149.309
C04781=1137.484,-23.477,-47.985,179.380,6.226,149.308
C04782=1137.479,-23.228,-47.997,179.383,6.227,149.308
C04783=1137.474,-22.978,-48.009,179.385,6.228,149.307
C04784=1137.468,-22.729,-48.022,179.387,6.228,149.307
C04785=1137.463,-22.479,-48.034,179.390,6.229,149.306
C04786=1137.458,-22.229,-48.045,179.392,6.230,149.306
C04787=1137.452,-21.979,-48.058,179.394,6.230,149.305
C04788=1137.448,-21.730,-48.069,179.397,6.231,149.305
C04789=1137.443,-21.480,-48.082,179.399,6.232,149.304
C04790=1137.437,-21.231,-48.094,179.401,6.232,149.303
C04791=1137.432,-20.981,-48.106,179.404,6.233,149.303
C04792=1137.427,-20.731,-48.118,179.406,6.234,149.302
C04793=1137.421,-20.482,-48.131,179.409,6.235,149.302
C04794=1137.416,-20.232,-48.143,179.411,6.236,149.301
C04795=1137.411,-19.983,-48.155,179.413,6.236,149.301
C04796=1137.405,-19.733,-48.167,179.416,6.237,149.300
C04797=1137.400,-19.483,-48.180,179.418,6.238,149.300
C04798=1137.395,-19.234,-48.192,179.421,6.238,149.299
C04799=1137.390,-18.984,-48.205,179.423,6.239,149.298
C04800=1137.385,-18.734,-48.217,179.425,6.240,149.298
C04801=1137.380,-18.484,-48.229,179.428,6.240,149.297
C04802=1137.374,-18.234,-48.241,179.430,6.241,149.297
C04803=1137.369,-17.985,-48.254,179.433,6.242,149.296
C04804=1137.364,-17.735,-48.266,179.436,6.243,149.296
C04805=1137.359,-17.486,-48.278,179.438,6.244,149.295
C04806=1137.354,-17.236,-48.291,179.440,6.244,149.295
C04807=1137.348,-16.987,-48.303,179.443,6.245,149.294
C04808=1137.343,-16.737,-48.315,179.445,6.246,149.294
C04809=1137.338,-16.487,-48.327,179.447,6.246,149.293
C04810=1137.333,-16.237,-48.340,179.450,6.247,149.292
C04811=1137.328,-15.988,-48.353,179.452,6.248,149.292
C04812=1137.323,-15.738,-48.365,179.455,6.249,149.291
C04813=1137.317,-15.489,-48.377,179.457,6.250,149.291
C04814=1137.312,-15.239,-48.390,179.459,6.250,149.290
C04815=1137.307,-14.989,-48.402,179.462,6.251,149.290
C04816=1137.302,-14.740,-48.414,179.464,6.252,149.289
C04817=1137.297,-14.490,-48.427,179.467,6.252,149.289
C04818=1137.292,-14.240,-48.439,179.469,6.253,149.288
C04819=1137.287,-13.991,-48.452,179.471,6.254,149.287
C04820=1137.282,-13.742,-48.464,179.474,6.255,149.287
C04821=1137.276,-13.492,-48.476,179.477,6.256,149.286
C04822=1137.271,-13.242,-48.489,179.479,6.256,149.286
C04823=1137.265,-12.993,-48.502,179.481,6.257,149.285
C04824=1137.261,-12.743,-48.515,179.484,6.258,149.285
C04825=1137.255,-12.493,-48.527,179.486,6.258,149.284
C04826=1137.250,-12.243,-48.540,179.488,6.259,149.284
C04827=1137.245,-11.994,-48.552,179.491,6.260,149.283
C04828=1137.240,-11.745,-48.565,179.494,6.261,149.283
C04829=1137.235,-11.495,-48.578,179.496,6.262,149.282
C04830=1137.230,-11.245,-48.590,179.498,6.262,149.281
C04831=1137.224,-10.995,-48.603,179.501,6.263,149.281
C04832=1137.219,-10.746,-48.615,179.503,6.264,149.280
C04833=1137.214,-10.496,-48.628,179.505,6.264,149.280
C04834=1137.209,-10.246,-48.641,179.508,6.266,149.279
C04835=1137.204,-9.997,-48.653,179.511,6.266,149.279
C04836=1137.199,-9.747,-48.665,179.513,6.267,149.278
C04837=1137.194,-9.498,-48.678,179.515,6.268,149.278
C04838=1137.188,-9.248,-48.692,179.518,6.269,149.277
C04839=1137.183,-8.998,-48.704,179.520,6.269,149.277
C04840=1137.178,-8.749,-48.717,179.522,6.270,149.276
C04841=1137.173,-8.500,-48.729,179.526,6.271,149.275
C04842=1137.168,-8.250,-48.742,179.528,6.272,149.275
C04843=1137.162,-7.999,-48.755,179.530,6.273,149.274
C04844=1137.157,-7.750,-48.767,179.533,6.273,149.274
C04845=1137.152,-7.501,-48.780,179.535,6.274,149.273
C04846=1137.147,-7.251,-48.793,179.537,6.275,149.273
C04847=1137.142,-7.001,-48.806,179.540,6.276,149.272
C04848=1137.136,-6.752,-48.819,179.542,6.277,149.272
C04849=1137.131,-6.502,-48.831,179.545,6.277,149.271
C04850=1137.127,-6.252,-48.844,179.547,6.278,149.270
C04851=1137.121,-6.003,-48.858,179.549,6.279,149.270
C04852=1137.116,-5.753,-48.870,179.553,6.280,149.269
C04853=1137.111,-5.504,-48.883,179.555,6.281,149.269
C04854=1137.105,-5.254,-48.896,179.557,6.282,149.268
C04855=1137.100,-5.005,-48.909,179.560,6.282,149.268
C04856=1137.095,-4.755,-48.922,179.562,6.283,149.267
C04857=1137.091,-4.505,-48.934,179.564,6.283,149.267
C04858=1137.085,-4.256,-48.948,179.567,6.285,149.266
C04859=1137.080,-4.006,-48.960,179.569,6.286,149.266
C04860=1137.075,-3.756,-48.973,179.572,6.286,149.265
C04861=1137.069,-3.507,-48.986,179.574,6.287,149.264
C04862=1137.064,-3.257,-48.999,179.576,6.288,149.264
C04863=1137.060,-3.007,-49.012,179.580,6.289,149.263
C04864=1137.054,-2.758,-49.025,179.582,6.290,149.263
C04865=1137.049,-2.508,-49.038,179.584,6.291,149.262
C04866=1137.044,-2.259,-49.051,179.587,6.291,149.262
C04867=1137.039,-2.009,-49.065,179.589,6.292,149.261
C04868=1137.034,-1.760,-49.077,179.592,6.293,149.261
C04869=1137.028,-1.510,-49.091,179.594,6.294,149.260
C04870=1137.023,-1.260,-49.103,179.597,6.295,149.260
C04871=1137.018,-1.011,-49.116,179.599,6.295,149.259
C04872=1137.013,-0.761,-49.130,179.601,6.296,149.258
C04873=1137.008,-0.511,-49.142,179.604,6.298,149.258
C04874=1137.002,-0.262,-49.156,179.607,6.298,149.257
C04875=1136.998,-0.012,-49.169,179.609,6.299,149.257
C04876=1136.992,0.237,-49.182,179.611,6.300,149.256
C04877=1136.987,0.487,-49.195,179.614,6.301,149.256
C04878=1136.982,0.737,-49.208,179.617,6.302,149.255
C04879=1136.977,1.006,-49.223,179.619,6.302,149.255
C04880=1136.970,1.275,-49.237,179.622,6.304,149.254
C04881=1136.965,1.545,-49.250,179.625,6.304,149.253
C04882=1136.960,1.815,-49.265,179.627,6.305,149.253
C04883=1136.955,2.064,-49.278,179.630,6.306,149.252
C04884=1136.949,2.314,-49.292,179.632,6.307,149.252
C04885=1136.945,2.563,-49.305,179.634,6.308,149.251
C04886=1136.939,2.813,-49.318,179.637,6.308,149.251
C04887=1136.934,3.063,-49.331,179.640,6.310,149.250
C04888=1136.928,3.312,-49.344,179.643,6.310,149.249
C04889=1136.924,3.562,-49.358,179.645,6.311,149.249
C04890=1136.918,3.811,-49.371,179.647,6.312,149.248
C04891=1136.914,4.061,-49.384,179.650,6.313,149.248
C04892=1136.908,4.310,-49.398,179.652,6.314,149.247
C04893=1136.904,4.560,-49.411,179.655,6.315,149.247
C04894=1136.898,4.810,-49.424,179.657,6.315,149.246
C04895=1136.893,5.059,-49.437,179.660,6.317,149.246
C04896=1136.888,5.309,-49.451,179.662,6.317,149.245
C04897=1136.883,5.558,-49.464,179.665,6.318,149.245
C04898=1136.878,5.808,-49.478,179.667,6.319,149.244
C04899=1136.872,6.058,-49.491,179.670,6.320,149.244
C04900=1136.868,6.307,-49.505,179.672,6.321,149.243
C04901=1136.862,6.557,-49.518,179.675,6.321,149.242
C04902=1136.857,6.807,-49.531,179.677,6.322,149.242
C04903=1136.852,7.056,-49.545,179.680,6.323,149.241
C04904=1136.846,7.306,-49.558,179.682,6.324,149.241
C04905=1136.842,7.555,-49.572,179.685,6.325,149.240
C04906=1136.836,7.805,-49.585,179.687,6.326,149.240
C04907=1136.831,8.054,-49.599,179.690,6.327,149.239
C04908=1136.826,8.304,-49.612,179.692,6.328,149.239
C04909=1136.821,8.553,-49.626,179.695,6.328,149.238
C04910=1136.816,8.803,-49.639,179.697,6.330,149.238
C04911=1136.811,9.052,-49.653,179.700,6.330,149.237
C04912=1136.805,9.302,-49.667,179.702,6.331,149.237
C04913=1136.801,9.552,-49.680,179.705,6.332,149.236
C04914=1136.795,9.801,-49.693,179.708,6.333,149.235
C04915=1136.791,10.051,-49.707,179.710,6.334,149.235
C04916=1136.785,10.300,-49.720,179.712,6.334,149.234
C04917=1136.780,10.550,-49.735,179.715,6.336,149.234
C04918=1136.774,10.800,-49.748,179.717,6.337,149.233
C04919=1136.770,11.049,-49.761,179.720,6.337,149.233
C04920=1136.764,11.299,-49.775,179.722,6.338,149.232
C04921=1136.759,11.549,-49.789,179.725,6.340,149.232
C04922=1136.755,11.798,-49.803,179.728,6.340,149.231
C04923=1136.749,12.048,-49.816,179.730,6.341,149.231
C04924=1136.744,12.297,-49.830,179.733,6.343,149.230
C04925=1136.739,12.547,-49.843,179.735,6.343,149.229
C04926=1136.734,12.796,-49.857,179.737,6.344,149.229
C04927=1136.729,13.045,-49.871,179.740,6.344,149.228
C04928=1136.723,13.296,-49.884,179.743,6.346,149.228
C04929=1136.719,13.545,-49.898,179.745,6.347,149.227
C04930=1136.714,13.794,-49.912,179.748,6.347,149.227
C04931=1136.708,14.044,-49.926,179.750,6.349,149.226
C04932=1136.703,14.293,-49.940,179.753,6.350,149.226
C04933=1136.698,14.543,-49.954,179.755,6.350,149.225
C04934=1136.693,14.793,-49.967,179.758,6.352,149.225
C04935=1136.688,15.042,-49.981,179.760,6.352,149.224
C04936=1136.683,15.292,-49.995,179.763,6.353,149.223
C04937=1136.678,15.542,-50.009,179.766,6.354,149.223
C04938=1136.672,15.791,-50.022,179.768,6.355,149.223
C04939=1136.668,16.041,-50.036,179.770,6.356,149.222
C04940=1136.663,16.290,-50.050,179.773,6.357,149.221
C04941=1136.657,16.539,-50.064,179.775,6.358,149.221
C04942=1136.652,16.790,-50.078,179.778,6.359,149.220
C04943=1136.647,17.039,-50.092,179.781,6.360,149.220
C04944=1136.642,17.288,-50.105,179.783,6.361,149.219
C04945=1136.637,17.538,-50.120,179.786,6.361,149.219
C04946=1136.632,17.787,-50.134,179.788,6.363,149.218
C04947=1136.626,18.037,-50.147,179.791,6.363,149.217
C04948=1136.622,18.287,-50.161,179.793,6.364,149.217
C04949=1136.617,18.536,-50.176,179.796,6.366,149.217
C04950=1136.611,18.785,-50.190,179.799,6.366,149.216
C04951=1136.606,19.035,-50.204,179.801,6.367,149.215
C04952=1136.602,19.285,-50.218,179.804,6.369,149.215
C04953=1136.596,19.534,-50.231,179.806,6.369,149.214
C04954=1136.591,19.784,-50.245,179.808,6.370,149.214
C04955=1136.586,20.034,-50.259,179.811,6.372,149.213
C04956=1136.581,20.283,-50.274,179.814,6.372,149.213
C04957=1136.576,20.532,-50.288,179.816,6.373,149.212
C04958=1136.571,20.782,-50.302,179.819,6.374,149.212
C04959=1136.566,21.032,-50.316,179.821,6.375,149.211
C04960=1136.560,21.281,-50.330,179.824,6.377,149.211
C04961=1136.555,21.531,-50.344,179.827,6.377,149.210
C04962=1136.550,21.780,-50.359,179.829,6.378,149.210
C04963=1136.545,22.030,-50.373,179.832,6.379,149.209
C04964=1136.540,22.279,-50.387,179.834,6.380,149.208
C04965=1136.535,22.529,-50.401,179.837,6.381,149.208
C04966=1136.530,22.778,-50.415,179.839,6.382,149.207
C04967=1136.525,23.028,-50.430,179.842,6.383,149.207
C04968=1136.520,23.278,-50.444,179.845,6.384,149.206
C04969=1136.514,23.527,-50.458,179.847,6.385,149.206
C04970=1136.509,23.776,-50.472,179.850,6.386,149.205
C04971=1136.504,24.026,-50.486,179.852,6.387,149.205
C04972=1136.499,24.276,-50.501,179.855,6.388,149.204
C04973=1136.494,24.525,-50.515,179.857,6.388,149.204
C04974=1136.489,24.775,-50.529,179.860,6.390,149.203
C04975=1136.484,25.024,-50.543,179.862,6.391,149.203
C04976=1136.479,25.274,-50.557,179.865,6.392,149.202
C04977=1136.474,25.524,-50.572,179.868,6.393,149.202
C04978=1136.469,25.773,-50.586,179.870,6.394,149.201
C04979=1136.464,26.022,-50.600,179.873,6.395,149.200
C04980=1136.459,26.272,-50.614,179.875,6.396,149.200
C04981=1136.454,26.521,-50.629,179.878,6.397,149.199
C04982=1136.449,26.771,-50.643,179.881,6.398,149.199
C04983=1136.443,27.041,-50.659,179.883,6.400,149.198
C04984=1136.438,27.310,-50.675,179.886,6.400,149.198
C04985=1136.432,27.578,-50.690,179.889,6.402,149.197
C04986=1136.427,27.847,-50.705,179.891,6.402,149.197
C04987=1136.422,28.097,-50.719,179.894,6.404,149.196
C04988=1136.416,28.346,-50.735,179.897,6.404,149.195
C04989=1136.411,28.596,-50.749,179.900,6.406,149.195
C04990=1136.406,28.846,-50.763,179.902,6.407,149.195
C04991=1136.401,29.095,-50.778,179.904,6.407,149.194
C04992=1136.396,29.344,-50.792,179.907,6.409,149.193
C04993=1136.391,29.593,-50.807,179.909,6.409,149.193
C04994=1136.386,29.843,-50.821,179.913,6.411,149.192
C04995=1136.380,30.093,-50.836,179.915,6.411,149.192
C04996=1136.376,30.343,-50.850,179.918,6.413,149.191
C04997=1136.371,30.592,-50.865,179.920,6.414,149.191
C04998=1136.366,30.842,-50.879,179.922,6.414,149.190
C04999=1136.361,31.091,-50.894,179.925,6.416,149.190
C05000=1136.356,31.341,-50.909,179.928,6.416,149.189
C05001=1136.351,31.590,-50.923,179.931,6.418,149.189
C05002=1136.345,31.839,-50.937,179.933,6.419,149.188
C05003=1136.340,32.089,-50.952,179.936,6.420,149.187
C05004=1136.335,32.338,-50.967,179.938,6.421,149.187
C05005=1136.330,32.588,-50.981,179.940,6.422,149.187
C05006=1136.325,32.837,-50.996,179.944,6.423,149.186
C05007=1136.320,33.087,-51.011,179.946,6.424,149.185
C05008=1136.315,33.337,-51.025,179.948,6.425,149.185
C05009=1136.310,33.586,-51.041,179.951,6.426,149.184
C05010=1136.305,33.836,-51.055,179.954,6.428,149.184
C05011=1136.300,34.085,-51.070,179.956,6.428,149.183
C05012=1136.295,34.335,-51.085,179.959,6.430,149.183
C05013=1136.290,34.585,-51.099,179.961,6.430,149.182
C05014=1136.285,34.834,-51.114,179.964,6.431,149.182
C05015=1136.280,35.084,-51.128,179.967,6.432,149.181
C05016=1136.275,35.333,-51.144,179.969,6.433,149.181
C05017=1136.270,35.583,-51.158,179.972,6.435,149.180
C05018=1136.265,35.832,-51.173,179.974,6.435,149.180
C05019=1136.259,36.082,-51.188,179.977,6.437,149.179
C05020=1136.255,36.331,-51.203,179.979,6.438,149.179
C05021=1136.249,36.581,-51.218,179.983,6.439,149.178
C05022=1136.244,36.830,-51.233,179.985,6.440,149.178
C05023=1136.239,37.080,-51.247,179.988,6.442,149.177
C05024=1136.234,37.329,-51.263,179.990,6.442,149.176
C05025=1136.229,37.579,-51.277,179.993,6.444,149.176
C05026=1136.224,37.828,-51.292,179.995,6.444,149.176
C05027=1136.219,38.078,-51.307,179.998,6.446,149.175
C05028=1136.214,38.327,-51.322,-180.000,6.447,149.174
C05029=1136.209,38.576,-51.337,-179.997,6.448,149.174
C05030=1136.204,38.826,-51.352,-179.994,6.449,149.173
C05031=1136.199,39.075,-51.367,-179.991,6.450,149.173
C05032=1136.193,39.325,-51.382,-179.989,6.451,149.172
C05033=1136.189,39.574,-51.397,-179.986,6.452,149.172
C05034=1136.183,39.824,-51.412,-179.984,6.453,149.171
C05035=1136.178,40.073,-51.426,-179.981,6.455,149.171
C05036=1136.173,40.323,-51.442,-179.978,6.455,149.170
C05037=1136.168,40.572,-51.457,-179.976,6.457,149.170
C05038=1136.163,40.822,-51.472,-179.973,6.458,149.169
C05039=1136.158,41.071,-51.487,-179.970,6.459,149.169
C05040=1136.153,41.320,-51.502,-179.968,6.460,149.168
C05041=1136.148,41.571,-51.517,-179.965,6.461,149.168
C05042=1136.144,41.820,-51.532,-179.963,6.462,149.167
C05043=1136.138,42.069,-51.548,-179.960,6.463,149.167
C05044=1136.133,42.319,-51.562,-179.958,6.464,149.166
C05045=1136.128,42.568,-51.578,-179.955,6.466,149.166
C05046=1136.123,42.818,-51.593,-179.952,6.466,149.165
C05047=1136.118,43.067,-51.608,-179.950,6.468,149.165
C05048=1136.112,43.317,-51.623,-179.947,6.469,149.164
C05049=1136.107,43.566,-51.638,-179.944,6.470,149.163
C05050=1136.103,43.816,-51.654,-179.942,6.471,149.163
C05051=1136.098,44.065,-51.669,-179.939,6.473,149.163
C05052=1136.093,44.315,-51.685,-179.937,6.473,149.162
C05053=1136.088,44.564,-51.699,-179.934,6.475,149.161
C05054=1136.082,44.814,-51.714,-179.932,6.475,149.161
C05055=1136.078,45.063,-51.729,-179.928,6.477,149.160
C05056=1136.072,45.312,-51.745,-179.926,6.478,149.160
C05057=1136.067,45.562,-51.761,-179.923,6.479,149.159
C05058=1136.063,45.811,-51.776,-179.921,6.480,149.159
C05059=1136.057,46.061,-51.791,-179.918,6.481,149.158
C05060=1136.052,46.311,-51.806,-179.916,6.482,149.158
C05061=1136.047,46.560,-51.821,-179.913,6.484,149.157
C05062=1136.042,46.810,-51.837,-179.910,6.485,149.157
C05063=1136.038,47.059,-51.852,-179.908,6.486,149.156
C05064=1136.032,47.309,-51.868,-179.905,6.487,149.156
C05065=1136.028,47.558,-51.883,-179.902,6.488,149.155
C05066=1136.022,47.807,-51.899,-179.900,6.490,149.155
C05067=1136.017,48.057,-51.915,-179.897,6.490,149.154
C05068=1136.013,48.306,-51.929,-179.894,6.492,149.154
C05069=1136.007,48.556,-51.945,-179.892,6.492,149.153
C05070=1136.002,48.805,-51.961,-179.889,6.494,149.153
C05071=1135.997,49.054,-51.976,-179.886,6.495,149.152
C05072=1135.993,49.304,-51.992,-179.884,6.496,149.152
C05073=1135.987,49.554,-52.007,-179.881,6.498,149.151
C05074=1135.983,49.803,-52.022,-179.879,6.499,149.151
C05075=1135.977,50.052,-52.038,-179.876,6.500,149.150
C05076=1135.972,50.302,-52.054,-179.874,6.501,149.150
C05077=1135.967,50.552,-52.069,-179.871,6.502,149.149
C05078=1135.962,50.801,-52.084,-179.868,6.504,149.148
C05079=1135.957,51.050,-52.100,-179.865,6.504,149.148
C05080=1135.952,51.300,-52.116,-179.863,6.506,149.148
C05081=1135.947,51.550,-52.131,-179.860,6.507,149.147
C05082=1135.942,51.799,-52.146,-179.857,6.508,149.146
C05083=1135.937,52.049,-52.162,-179.855,6.509,149.146
C05084=1135.932,52.298,-52.178,-179.852,6.511,149.146
C05085=1135.927,52.548,-52.194,-179.849,6.512,149.145
C05086=1135.922,52.796,-52.209,-179.847,6.513,149.144
C05087=1135.917,53.066,-52.226,-179.844,6.514,149.144
C05088=1135.911,53.334,-52.243,-179.841,6.516,149.143
C05089=1135.906,53.603,-52.260,-179.838,6.517,149.143
C05090=1135.900,53.871,-52.277,-179.836,6.518,149.142
C05091=1135.895,54.121,-52.293,-179.833,6.519,149.142
C05092=1135.890,54.371,-52.309,-179.830,6.521,149.141
C05093=1135.886,54.619,-52.324,-179.827,6.522,149.141
C05094=1135.880,54.869,-52.340,-179.825,6.523,149.140
C05095=1135.876,55.119,-52.356,-179.822,6.524,149.140
C05096=1135.870,55.368,-52.371,-179.819,6.525,149.139
C05097=1135.865,55.617,-52.388,-179.816,6.527,149.139
C05098=1135.860,55.867,-52.404,-179.814,6.528,149.138
C05099=1135.855,56.117,-52.419,-179.812,6.529,149.138
C05100=1135.850,56.366,-52.434,-179.809,6.530,149.137
C05101=1135.846,56.615,-52.451,-179.806,6.531,149.137
C05102=1135.840,56.865,-52.466,-179.803,6.533,149.136
C05103=1135.835,57.114,-52.482,-179.801,6.534,149.136
C05104=1135.831,57.363,-52.499,-179.798,6.535,149.135
C05105=1135.825,57.613,-52.514,-179.796,6.536,149.135
C05106=1135.820,57.863,-52.530,-179.793,6.538,149.134
C05107=1135.815,58.112,-52.547,-179.790,6.539,149.134
C05108=1135.810,58.361,-52.562,-179.788,6.540,149.133
C05109=1135.805,58.611,-52.578,-179.785,6.541,149.133
C05110=1135.800,58.860,-52.594,-179.782,6.543,149.132
C05111=1135.795,59.110,-52.610,-179.780,6.544,149.132
C05112=1135.790,59.359,-52.626,-179.777,6.545,149.131
C05113=1135.785,59.608,-52.642,-179.774,6.547,149.131
C05114=1135.780,59.858,-52.658,-179.771,6.547,149.130
C05115=1135.775,60.107,-52.675,-179.769,6.549,149.130
C05116=1135.770,60.357,-52.690,-179.766,6.550,149.129
C05117=1135.765,60.607,-52.706,-179.764,6.551,149.129
C05118=1135.760,60.856,-52.723,-179.760,6.553,149.128
C05119=1135.755,61.106,-52.738,-179.758,6.554,149.128
C05120=1135.750,61.354,-52.755,-179.756,6.555,149.127
C05121=1135.745,61.604,-52.771,-179.752,6.556,149.127
C05122=1135.740,61.853,-52.787,-179.750,6.557,149.126
C05123=1135.735,62.103,-52.803,-179.747,6.559,149.126
C05124=1135.730,62.352,-52.819,-179.745,6.561,149.125
C05125=1135.725,62.602,-52.835,-179.742,6.561,149.125
C05126=1135.720,62.851,-52.851,-179.739,6.563,149.124
C05127=1135.715,63.101,-52.867,-179.737,6.564,149.124
C05128=1135.710,63.350,-52.884,-179.734,6.565,149.123
C05129=1135.706,63.599,-52.900,-179.731,6.566,149.123
C05130=1135.701,63.849,-52.916,-179.728,6.568,149.122
C05131=1135.696,64.098,-52.933,-179.726,6.569,149.122
C05132=1135.691,64.348,-52.948,-179.723,6.571,149.121
C05133=1135.686,64.597,-52.965,-179.720,6.572,149.121
C05134=1135.680,64.846,-52.982,-179.718,6.573,149.120
C05135=1135.676,65.096,-52.998,-179.715,6.574,149.120
C05136=1135.670,65.345,-53.014,-179.713,6.576,149.119
C05137=1135.666,65.595,-53.030,-179.710,6.576,149.119
C05138=1135.661,65.844,-53.046,-179.707,6.578,149.118
C05139=1135.656,66.093,-53.063,-179.704,6.580,149.118
C05140=1135.651,66.343,-53.079,-179.702,6.581,149.117
C05141=1135.646,66.592,-53.095,-179.699,6.582,149.117
C05142=1135.641,66.842,-53.112,-179.696,6.584,149.116
C05143=1135.636,67.091,-53.129,-179.694,6.585,149.116
C05144=1135.631,67.341,-53.145,-179.691,6.586,149.115
C05145=1135.626,67.590,-53.161,-179.688,6.587,149.115
C05146=1135.622,67.839,-53.178,-179.685,6.589,149.114
C05147=1135.615,68.089,-53.194,-179.683,6.590,149.114
C05148=1135.611,68.339,-53.211,-179.680,6.591,149.113
C05149=1135.607,68.588,-53.227,-179.677,6.593,149.113
C05150=1135.601,68.837,-53.243,-179.675,6.594,149.112
C05151=1135.597,69.086,-53.260,-179.672,6.595,149.112
C05152=1135.591,69.336,-53.276,-179.670,6.597,149.111
C05153=1135.586,69.585,-53.293,-179.666,6.598,149.111
C05154=1135.582,69.835,-53.310,-179.664,6.599,149.110
C05155=1135.576,70.084,-53.327,-179.661,6.601,149.110
C05156=1135.572,70.334,-53.343,-179.659,6.602,149.110
C05157=1135.566,70.583,-53.359,-179.656,6.603,149.109
C05158=1135.562,70.832,-53.376,-179.653,6.604,149.108
C05159=1135.556,71.082,-53.393,-179.651,6.606,149.108
C05160=1135.551,71.331,-53.409,-179.648,6.608,149.108
C05161=1135.547,71.580,-53.426,-179.645,6.608,149.107
C05162=1135.542,71.830,-53.443,-179.642,6.610,149.106
C05163=1135.537,72.079,-53.459,-179.640,6.611,149.106
C05164=1135.532,72.329,-53.476,-179.638,6.612,149.106
C05165=1135.527,72.578,-53.493,-179.634,6.614,149.105
C05166=1135.522,72.827,-53.510,-179.632,6.615,149.105
C05167=1135.517,73.077,-53.526,-179.629,6.617,149.104
C05168=1135.512,73.327,-53.543,-179.627,6.618,149.104
C05169=1135.507,73.576,-53.559,-179.623,6.619,149.103
C05170=1135.502,73.825,-53.576,-179.621,6.621,149.103
C05171=1135.497,74.075,-53.593,-179.618,6.622,149.102
C05172=1135.492,74.324,-53.609,-179.616,6.623,149.102
C05173=1135.488,74.573,-53.626,-179.613,6.625,149.101
C05174=1135.482,74.823,-53.643,-179.610,6.626,149.101
C05175=1135.477,75.072,-53.660,-179.607,6.628,149.100
C05176=1135.472,75.321,-53.678,-179.605,6.629,149.100
C05177=1135.468,75.571,-53.694,-179.602,6.630,149.099
C05178=1135.463,75.820,-53.711,-179.599,6.632,149.099
C05179=1135.458,76.069,-53.728,-179.596,6.633,149.098
C05180=1135.453,76.319,-53.744,-179.594,6.634,149.098
C05181=1135.448,76.568,-53.762,-179.591,6.636,149.097
C05182=1135.443,76.817,-53.778,-179.589,6.637,149.097
C05183=1135.438,77.067,-53.795,-179.585,6.639,149.096
C05184=1135.433,77.316,-53.812,-179.583,6.640,149.096
C05185=1135.428,77.566,-53.829,-179.580,6.641,149.095
C05186=1135.423,77.814,-53.846,-179.578,6.643,149.095
C05187=1135.418,78.064,-53.863,-179.575,6.644,149.095
C05188=1135.413,78.314,-53.880,-179.572,6.646,149.094
C05189=1135.408,78.564,-53.897,-179.570,6.647,149.093
C05190=1135.403,78.812,-53.914,-179.567,6.648,149.093
C05191=1135.398,79.081,-53.932,-179.564,6.650,149.093
C05192=1135.393,79.350,-53.951,-179.561,6.651,149.092
C05193=1135.387,79.618,-53.969,-179.558,6.653,149.092
C05194=1135.382,79.887,-53.988,-179.555,6.654,149.091
C05195=1135.377,80.136,-54.005,-179.552,6.656,149.090
C05196=1135.372,80.385,-54.022,-179.549,6.657,149.090
C05197=1135.367,80.634,-54.038,-179.547,6.659,149.090
C05198=1135.362,80.883,-54.056,-179.544,6.660,149.089
C05199=1135.357,81.133,-54.074,-179.541,6.661,149.089
C05200=1135.353,81.383,-54.090,-179.539,6.663,149.088
C05201=1135.347,81.632,-54.108,-179.536,6.665,149.088
C05202=1135.343,81.881,-54.125,-179.533,6.666,149.087
C05203=1135.337,82.130,-54.142,-179.531,6.667,149.087
C05204=1135.332,82.380,-54.159,-179.528,6.668,149.086
C05205=1135.328,82.629,-54.177,-179.525,6.670,149.086
C05206=1135.323,82.879,-54.194,-179.522,6.672,149.085
C05207=1135.318,83.128,-54.211,-179.519,6.673,149.085
C05208=1135.313,83.377,-54.228,-179.517,6.674,149.084
C05209=1135.308,83.627,-54.245,-179.514,6.675,149.084
C05210=1135.303,83.875,-54.263,-179.511,6.677,149.083
C05211=1135.298,84.125,-54.280,-179.509,6.679,149.083
C05212=1135.293,84.375,-54.297,-179.506,6.680,149.083
C05213=1135.289,84.624,-54.315,-179.503,6.682,149.082
C05214=1135.284,84.874,-54.332,-179.500,6.683,149.081
C05215=1135.279,85.123,-54.350,-179.498,6.684,149.081
C05216=1135.274,85.372,-54.367,-179.495,6.686,149.081
C05217=1135.269,85.621,-54.384,-179.492,6.688,149.080
C05218=1135.263,85.871,-54.401,-179.489,6.689,149.080
C05219=1135.258,86.120,-54.419,-179.487,6.691,149.079
C05220=1135.254,86.369,-54.436,-179.484,6.691,149.079
C05221=1135.249,86.619,-54.454,-179.481,6.693,149.078
C05222=1135.244,86.868,-54.471,-179.479,6.695,149.078
C05223=1135.239,87.117,-54.489,-179.476,6.696,149.077
C05224=1135.234,87.367,-54.506,-179.473,6.698,149.077
C05225=1135.230,87.616,-54.524,-179.470,6.700,149.077
C05226=1135.224,87.866,-54.541,-179.468,6.700,149.076
C05227=1135.219,88.115,-54.559,-179.465,6.702,149.075
C05228=1135.215,88.364,-54.577,-179.462,6.703,149.075
C05229=1135.210,88.614,-54.594,-179.460,6.705,149.075
C05230=1135.205,88.863,-54.612,-179.457,6.707,149.074
C05231=1135.200,89.113,-54.629,-179.454,6.708,149.074
C05232=1135.195,89.362,-54.647,-179.451,6.710,149.073
C05233=1135.190,89.611,-54.665,-179.449,6.711,149.073
C05234=1135.186,89.861,-54.682,-179.446,6.712,149.072
C05235=1135.181,90.110,-54.700,-179.443,6.714,149.072
C05236=1135.176,90.359,-54.718,-179.440,6.716,149.071
C05237=1135.171,90.609,-54.735,-179.438,6.717,149.071
C05238=1135.166,90.858,-54.753,-179.434,6.719,149.070
C05239=1135.161,91.107,-54.771,-179.432,6.720,149.070
C05240=1135.156,91.356,-54.789,-179.429,6.722,149.070
C05241=1135.151,91.606,-54.806,-179.427,6.723,149.069
C05242=1135.146,91.855,-54.824,-179.424,6.724,149.069
C05243=1135.142,92.104,-54.842,-179.421,6.726,149.068
C05244=1135.137,92.353,-54.860,-179.418,6.727,149.068
C05245=1135.131,92.603,-54.877,-179.415,6.729,149.067
C05246=1135.127,92.852,-54.895,-179.413,6.731,149.067
C05247=1135.122,93.101,-54.913,-179.410,6.732,149.066
C05248=1135.117,93.351,-54.931,-179.407,6.734,149.066
C05249=1135.111,93.600,-54.948,-179.404,6.736,149.066
C05250=1135.107,93.850,-54.966,-179.402,6.737,149.065
C05251=1135.102,94.099,-54.984,-179.399,6.738,149.064
C05252=1135.097,94.348,-55.002,-179.396,6.739,149.064
C05253=1135.092,94.597,-55.020,-179.394,6.741,149.064
C05254=1135.087,94.846,-55.038,-179.391,6.743,149.063
C05255=1135.082,95.095,-55.056,-179.388,6.744,149.063
C05256=1135.077,95.346,-55.074,-179.385,6.746,149.062
C05257=1135.072,95.595,-55.092,-179.383,6.748,149.062
C05258=1135.068,95.844,-55.109,-179.379,6.749,149.061
C05259=1135.063,96.093,-55.127,-179.377,6.751,149.061
C05260=1135.058,96.343,-55.145,-179.374,6.752,149.060
C05261=1135.053,96.592,-55.163,-179.372,6.753,149.060
C05262=1135.048,96.841,-55.181,-179.369,6.755,149.060
C05263=1135.043,97.090,-55.199,-179.366,6.757,149.059
C05264=1135.038,97.339,-55.217,-179.364,6.758,149.059
C05265=1135.034,97.589,-55.236,-179.361,6.760,149.058
C05266=1135.029,97.838,-55.254,-179.358,6.761,149.058
C05267=1135.024,98.088,-55.272,-179.355,6.763,149.057
C05268=1135.019,98.337,-55.290,-179.352,6.765,149.057
C05269=1135.014,98.586,-55.308,-179.349,6.766,149.056
C05270=1135.009,98.835,-55.326,-179.347,6.768,149.056
C05271=1135.004,99.085,-55.344,-179.344,6.770,149.056
C05272=1134.999,99.334,-55.363,-179.341,6.771,149.055
C05273=1134.994,99.584,-55.381,-179.338,6.773,149.055
C05274=1134.989,99.833,-55.398,-179.335,6.774,149.054
C05275=1134.985,100.082,-55.416,-179.333,6.776,149.054
C05276=1134.980,100.331,-55.435,-179.330,6.777,149.053
C05277=1134.976,100.580,-55.454,-179.328,6.778,149.053
C05278=1134.971,100.830,-55.471,-179.325,6.780,149.053
C05279=1134.965,101.079,-55.490,-179.322,6.782,149.052
C05280=1134.960,101.328,-55.508,-179.319,6.783,149.052
C05281=1134.955,101.577,-55.526,-179.317,6.785,149.051
C05282=1134.951,101.827,-55.544,-179.314,6.787,149.051
C05283=1134.946,102.076,-55.563,-179.311,6.788,149.050
C05284=1134.941,102.325,-55.582,-179.308,6.790,149.050
C05285=1134.936,102.575,-55.600,-179.305,6.791,149.049
C05286=1134.931,102.824,-55.618,-179.303,6.793,149.049
C05287=1134.927,103.074,-55.636,-179.300,6.795,149.049
C05288=1134.921,103.322,-55.655,-179.297,6.796,149.048
C05289=1134.916,103.572,-55.673,-179.294,6.798,149.048
C05290=1134.912,103.822,-55.692,-179.292,6.800,149.047
C05291=1134.907,104.071,-55.710,-179.289,6.801,149.047
C05292=1134.902,104.320,-55.729,-179.286,6.803,149.046
C05293=1134.897,104.569,-55.747,-179.283,6.804,149.046
C05294=1134.892,104.819,-55.765,-179.280,6.806,149.045
C05295=1134.887,105.087,-55.786,-179.277,6.808,149.045
C05296=1134.882,105.355,-55.805,-179.275,6.809,149.045
C05297=1134.877,105.623,-55.825,-179.271,6.812,149.044
C05298=1134.871,105.892,-55.845,-179.268,6.813,149.044
C05299=1134.867,106.141,-55.864,-179.265,6.815,149.043
C05300=1134.861,106.390,-55.882,-179.263,6.817,149.043
C05301=1134.856,106.640,-55.900,-179.260,6.818,149.042
C05302=1134.852,106.889,-55.919,-179.257,6.820,149.042
C05303=1134.847,107.138,-55.938,-179.254,6.822,149.042
C05304=1134.842,107.387,-55.957,-179.252,6.823,149.041
C05305=1134.838,107.637,-55.975,-179.249,6.825,149.041
C05306=1134.832,107.886,-55.994,-179.246,6.827,149.040
C05307=1134.828,108.135,-56.012,-179.244,6.828,149.040
C05308=1134.823,108.385,-56.031,-179.241,6.830,149.039
C05309=1134.818,108.634,-56.050,-179.238,6.832,149.039
C05310=1134.813,108.883,-56.068,-179.235,6.833,149.038
C05311=1134.808,109.132,-56.088,-179.232,6.835,149.038
C05312=1134.803,109.381,-56.106,-179.229,6.836,149.038
C05313=1134.799,109.630,-56.124,-179.227,6.838,149.037
C05314=1134.794,109.880,-56.143,-179.224,6.840,149.037
C05315=1134.789,110.129,-56.162,-179.221,6.841,149.036
C05316=1134.784,110.379,-56.181,-179.218,6.843,149.036
C05317=1134.779,110.627,-56.199,-179.216,6.845,149.036
C05318=1134.774,110.876,-56.219,-179.213,6.846,149.035
C05319=1134.770,111.126,-56.237,-179.210,6.848,149.035
C05320=1134.764,111.375,-56.256,-179.207,6.850,149.034
C05321=1134.760,111.625,-56.275,-179.205,6.851,149.034
C05322=1134.755,111.874,-56.294,-179.202,6.853,149.034
C05323=1134.750,112.122,-56.313,-179.199,6.855,149.033
C05324=1134.745,112.373,-56.332,-179.197,6.856,149.033
C05325=1134.741,112.621,-56.350,-179.194,6.858,149.032
C05326=1134.736,112.871,-56.370,-179.191,6.860,149.032
C05327=1134.731,113.120,-56.388,-179.188,6.861,149.031
C05328=1134.726,113.369,-56.408,-179.185,6.863,149.031
C05329=1134.722,113.618,-56.426,-179.182,6.864,149.030
C05330=1134.716,113.868,-56.445,-179.180,6.866,149.030
C05331=1134.711,114.117,-56.465,-179.176,6.869,149.030
C05332=1134.707,114.366,-56.483,-179.174,6.870,149.029
C05333=1134.701,114.616,-56.502,-179.171,6.872,149.029
C05334=1134.697,114.864,-56.521,-179.168,6.874,149.028
C05335=1134.692,115.114,-56.541,-179.165,6.875,149.028
C05336=1134.687,115.363,-56.560,-179.163,6.877,149.028
C05337=1134.683,115.612,-56.579,-179.160,6.879,149.027
C05338=1134.677,115.862,-56.598,-179.157,6.880,149.027
C05339=1134.673,116.111,-56.617,-179.155,6.882,149.026
C05340=1134.668,116.360,-56.636,-179.152,6.884,149.026
C05341=1134.663,116.609,-56.656,-179.149,6.885,149.026
C05342=1134.658,116.858,-56.674,-179.146,6.887,149.025
C05343=1134.653,117.108,-56.693,-179.144,6.889,149.025
C05344=1134.648,117.357,-56.712,-179.141,6.890,149.024
C05345=1134.644,117.606,-56.732,-179.138,6.893,149.024
C05346=1134.639,117.855,-56.751,-179.135,6.895,149.024
C05347=1134.634,118.105,-56.770,-179.132,6.896,149.023
C05348=1134.630,118.354,-56.790,-179.129,6.898,149.023
C05349=1134.625,118.603,-56.809,-179.127,6.900,149.022
C05350=1134.620,118.852,-56.828,-179.124,6.901,149.022
C05351=1134.614,119.101,-56.848,-179.121,6.903,149.022
C05352=1134.610,119.350,-56.867,-179.118,6.905,149.021
C05353=1134.605,119.599,-56.886,-179.116,6.906,149.021
C05354=1134.600,119.849,-56.906,-179.113,6.908,149.020
C05355=1134.596,120.097,-56.924,-179.110,6.910,149.020
C05356=1134.591,120.347,-56.944,-179.107,6.912,149.020
C05357=1134.586,120.596,-56.964,-179.104,6.914,149.019
C05358=1134.581,120.845,-56.983,-179.101,6.916,149.019
C05359=1134.576,121.095,-57.003,-179.099,6.917,149.018
C05360=1134.572,121.343,-57.021,-179.096,6.919,149.018
C05361=1134.567,121.593,-57.041,-179.093,6.921,149.017
C05362=1134.562,121.843,-57.061,-179.091,6.922,149.017
C05363=1134.557,122.091,-57.080,-179.088,6.924,149.017
C05364=1134.552,122.341,-57.100,-179.084,6.927,149.016
C05365=1134.548,122.590,-57.119,-179.082,6.928,149.016
C05366=1134.543,122.839,-57.138,-179.079,6.930,149.015
C05367=1134.538,123.089,-57.158,-179.076,6.932,149.015
C05368=1134.533,123.338,-57.177,-179.074,6.933,149.015
C05369=1134.528,123.587,-57.197,-179.071,6.935,149.014
C05370=1134.523,123.836,-57.217,-179.068,6.937,149.014
C05371=1134.519,124.085,-57.236,-179.065,6.938,149.013
C05372=1134.514,124.334,-57.255,-179.062,6.941,149.013
C05373=1134.509,124.584,-57.275,-179.059,6.943,149.013
C05374=1134.505,124.833,-57.295,-179.057,6.944,149.012
C05375=1134.500,125.082,-57.315,-179.054,6.946,149.012
C05376=1134.495,125.331,-57.334,-179.051,6.948,149.011
C05377=1134.490,125.581,-57.354,-179.048,6.949,149.011
C05378=1134.485,125.830,-57.373,-179.046,6.951,149.011
C05379=1134.480,126.079,-57.394,-179.042,6.953,149.010
C05380=1134.476,126.328,-57.413,-179.040,6.955,149.010
C05381=1134.471,126.577,-57.432,-179.037,6.957,149.010
C05382=1134.466,126.826,-57.452,-179.034,6.959,149.009
C05383=1134.462,127.075,-57.472,-179.031,6.960,149.009
C05384=1134.457,127.325,-57.492,-179.029,6.962,149.008
C05385=1134.452,127.573,-57.512,-179.025,6.964,149.008
C05386=1134.447,127.823,-57.531,-179.023,6.966,149.008
C05387=1134.442,128.072,-57.551,-179.020,6.968,149.007
C05388=1134.438,128.321,-57.571,-179.017,6.969,149.007
C05389=1134.433,128.570,-57.591,-179.015,6.971,149.007
C05390=1134.428,128.820,-57.610,-179.012,6.973,149.006
C05391=1134.424,129.068,-57.631,-179.009,6.976,149.006
C05392=1134.419,129.318,-57.650,-179.006,6.977,149.005
C05393=1134.414,129.566,-57.670,-179.004,6.979,149.005
C05394=1134.408,129.816,-57.691,-179.001,6.981,149.005
C05395=1134.404,130.066,-57.710,-178.998,6.982,149.004
C05396=1134.399,130.315,-57.731,-178.995,6.984,149.004
C05397=1134.394,130.564,-57.750,-178.992,6.987,149.003
C05398=1134.389,130.813,-57.770,-178.989,6.988,149.003
C05399=1134.384,131.081,-57.791,-178.987,6.990,149.003
C05400=1134.379,131.350,-57.813,-178.983,6.992,149.002
C05401=1134.374,131.618,-57.835,-178.981,6.994,149.002
C05402=1134.368,131.887,-57.857,-178.977,6.997,149.001
C05403=1134.364,132.136,-57.877,-178.974,6.998,149.001
C05404=1134.359,132.386,-57.897,-178.972,7.000,149.001
C05405=1134.355,132.635,-57.917,-178.969,7.002,149.000
C05406=1134.350,132.883,-57.936,-178.966,7.003,149.000
C05407=1134.345,133.132,-57.957,-178.963,7.006,148.999
C05408=1134.340,133.382,-57.978,-178.960,7.008,148.999
C05409=1134.335,133.631,-57.997,-178.958,7.009,148.999
C05410=1134.331,133.880,-58.018,-178.955,7.011,148.998
C05411=1134.326,134.130,-58.037,-178.952,7.013,148.998
C05412=1134.322,134.379,-58.058,-178.949,7.015,148.998
C05413=1134.317,134.628,-58.078,-178.947,7.017,148.997
C05414=1134.311,134.877,-58.098,-178.944,7.019,148.997
C05415=1134.307,135.126,-58.118,-178.941,7.021,148.997
C05416=1134.302,135.375,-58.139,-178.938,7.023,148.996
C05417=1134.297,135.624,-58.158,-178.935,7.025,148.996
C05418=1134.292,135.874,-58.179,-178.932,7.027,148.995
C05419=1134.288,136.123,-58.200,-178.930,7.028,148.995
C05420=1134.283,136.371,-58.220,-178.927,7.030,148.995
C05421=1134.279,136.621,-58.240,-178.924,7.032,148.994
C05422=1134.273,136.870,-58.261,-178.921,7.034,148.994
C05423=1134.269,137.119,-58.281,-178.919,7.036,148.994
C05424=1134.264,137.367,-58.301,-178.916,7.038,148.993
C05425=1134.260,137.616,-58.321,-178.913,7.040,148.993
C05426=1134.254,137.866,-58.342,-178.910,7.042,148.992
C05427=1134.250,138.115,-58.362,-178.907,7.044,148.992
C05428=1134.245,138.364,-58.382,-178.904,7.045,148.992
C05429=1134.240,138.613,-58.403,-178.901,7.048,148.991
C05430=1134.236,138.862,-58.424,-178.898,7.050,148.991
C05431=1134.231,139.111,-58.444,-178.896,7.051,148.991
C05432=1134.226,139.361,-58.464,-178.893,7.053,148.990
C05433=1134.221,139.610,-58.485,-178.890,7.056,148.990
C05434=1134.217,139.859,-58.505,-178.887,7.058,148.990
C05435=1134.212,140.108,-58.526,-178.885,7.059,148.989
C05436=1134.207,140.357,-58.546,-178.882,7.061,148.989
C05437=1134.202,140.607,-58.567,-178.879,7.063,148.988
C05438=1134.198,140.856,-58.588,-178.876,7.065,148.988
C05439=1134.193,141.104,-58.608,-178.873,7.067,148.988
C05440=1134.188,141.354,-58.629,-178.870,7.070,148.987
C05441=1134.183,141.603,-58.649,-178.868,7.071,148.987
C05442=1134.178,141.852,-58.670,-178.865,7.073,148.987
C05443=1134.174,142.101,-58.691,-178.862,7.075,148.986
C05444=1134.169,142.350,-58.712,-178.859,7.077,148.986
C05445=1134.164,142.599,-58.732,-178.856,7.079,148.986
C05446=1134.160,142.848,-58.753,-178.853,7.081,148.985
C05447=1134.155,143.097,-58.773,-178.851,7.084,148.985
C05448=1134.150,143.346,-58.794,-178.848,7.085,148.985
C05449=1134.146,143.596,-58.815,-178.845,7.087,148.984
C05450=1134.141,143.845,-58.836,-178.842,7.089,148.984
C05451=1134.136,144.094,-58.857,-178.839,7.091,148.983
C05452=1134.132,144.343,-58.878,-178.836,7.093,148.983
C05453=1134.127,144.592,-58.899,-178.834,7.095,148.983
C05454=1134.122,144.841,-58.919,-178.831,7.097,148.983
C05455=1134.117,145.090,-58.940,-178.828,7.099,148.982
C05456=1134.112,145.340,-58.961,-178.825,7.101,148.982
C05457=1134.108,145.588,-58.981,-178.822,7.103,148.981
C05458=1134.102,145.838,-59.002,-178.819,7.105,148.981
C05459=1134.098,146.086,-59.023,-178.817,7.107,148.981
C05460=1134.094,146.336,-59.045,-178.814,7.109,148.980
C05461=1134.089,146.585,-59.065,-178.811,7.111,148.980
C05462=1134.084,146.834,-59.086,-178.808,7.113,148.980
C05463=1134.079,147.083,-59.108,-178.806,7.115,148.979
C05464=1134.075,147.332,-59.128,-178.802,7.117,148.979
C05465=1134.070,147.581,-59.149,-178.800,7.119,148.979
C05466=1134.065,147.830,-59.169,-178.797,7.121,148.978
C05467=1134.061,148.079,-59.191,-178.794,7.123,148.978
C05468=1134.056,148.329,-59.212,-178.791,7.125,148.978
C05469=1134.051,148.578,-59.233,-178.789,7.127,148.977
C05470=1134.046,148.826,-59.254,-178.786,7.130,148.977
C05471=1134.041,149.075,-59.275,-178.783,7.131,148.977
C05472=1134.037,149.324,-59.296,-178.780,7.133,148.976
C05473=1134.032,149.574,-59.318,-178.777,7.136,148.976
C05474=1134.027,149.823,-59.339,-178.774,7.137,148.976
C05475=1134.023,150.072,-59.359,-178.772,7.139,148.975
C05476=1134.018,150.321,-59.381,-178.769,7.142,148.975
C05477=1134.013,150.570,-59.402,-178.766,7.144,148.975
